// TIA Portal project "Project1500" (V15.1)

(* hardware
DEVICE "S71500/ET200MP station_1"  S7-1500 station
   slot 0: "Rail_0"  Rack  6ES7 590-1***0-0AA0
   slot 1: "PLC_1"  CPU 1515-2 PN  6ES7 515-2AM01-0AB0  V2.6
      slot 3: "CPU display_1"  6ES7591-1BA00-0AA0
*)

// ===== PLC "PLC_1"  CPU 1515-2 PN =====

VAR_GLOBAL   // PLC tag table "Default tag table"
   "Clock_Byte" AT %MB90 : Byte;
   "Clock_10Hz" AT %M90.0 : Bool;
   "Clock_5Hz" AT %M90.1 : Bool;
   "Clock_2.5Hz" AT %M90.2 : Bool;
   "Clock_2Hz" AT %M90.3 : Bool;
   "Clock_1.25Hz" AT %M90.4 : Bool;
   "Clock_1Hz" AT %M90.5 : Bool;
   "Clock_0.625Hz" AT %M90.6 : Bool;
   "Clock_0.5Hz" AT %M90.7 : Bool;
END_VAR

VAR_GLOBAL   // PLC tag table "1AInputs"
   "PLC_AI_CH0" AT %IW64 : Int;   // Резерв
   "PLC_AI_CH1" AT %IW66 : Int;   // Резерв
   "A2_AI_CH0" AT %IW96 : Int;   // Разрежение на газоходе перед циклоном (Элемер-100-ДВ-1231М)
   "A2_AI_CH1" AT %IW98 : Int;   // Разрежение на газоходе перед рукавным фильтром (Элемер-100-ДВ-1231М)
   "A2_AI_CH2" AT %IW100 : Int;   // Разрежение на газоходе после рукавного фильтра (Элемер-100-ДВ-1231М)
   "A2_AI_CH3" AT %IW102 : Int;   // Давление на грубопроводе сжатого воздуха на входе в шатер рукавного фильтра (Элемер-100-ДИ-1150)
   "A2_AI_CH4" AT %IW104 : Int;   // Концентрация CO (Газоанализатор 503б)
   "A2_AI_CH5" AT %IW106 : Int;   // Концентрация SO2 (Газоанализатор 503б)
   "A2_AI_CH6" AT %IW108 : Int;   // Концентрация NOx (Газоанализатор 503б)
   "A2_AI_CH7" AT %IW110 : Int;   // Концентрация CO2 (Газоанализатор 503б)
   "A3_AI_CH0" AT %IW112 : Int;   // Концентрация O2 (Газоанализатор 503б)
   "A3_AI_CH1" AT %IW114 : Int;   // Расход пылегазовой смеси (Анализатор 303в)
   "A3_AI_CH2" AT %IW116 : Int;   // Концентрация пыли (Пылемер 403в)
   "A3_AI_CH3" AT %IW118 : Int;   // Положение: клапан регулирующий для аспирации 1M
   "A3_AI_CH4" AT %IW120 : Int;   // Контроль тока двигателя (Шкаф преобразователя частоты ШПЧ1)
   "A3_AI_CH5" AT %IW122 : Int;   // Контроль скорости двигателя (Шкаф преобразователя частоты ШПЧ1)
   "A3_AI_CH6" AT %IW124 : Int;   // Резерв
   "A3_AI_CH7" AT %IW126 : Int;   // Резерв
   "A4_AI_CH0" AT %IW128 : Int;   // Дымосос 1. Вибрация переднего подшипника вентилятора X-направления
   "A4_AI_CH1" AT %IW130 : Int;   // Дымосос 1. Вибрация переднего подшипника вентилятора Y-направления
   "A4_AI_CH2" AT %IW132 : Int;   // Дымосос 1. Вибрация заднего подшипника вентилятора X-направления
   "A4_AI_CH3" AT %IW134 : Int;   // Дымосос 1. Вибрация заднего подшипника вентилятора Y-направления
   "A4_AI_CH4" AT %IW136 : Int;   // Резерв
   "A4_AI_CH5" AT %IW138 : Int;   // Резерв
   "A4_AI_CH6" AT %IW140 : Int;   // Резерв
   "A4_AI_CH7" AT %IW142 : Int;   // Резерв
   "A5_AI_CH0" AT %IW144 : Int;   // Дымосос 1. Температура переднего подшипника вентилятора (Термопреобр. сопротивления TC-1088-Pt100)
   "A5_AI_CH1" AT %IW146 : Int;   // Дымосос 1. Температура заднего подшипника вентилятора (Термопреобр. сопротивления TC-1088-Pt100)
   "A5_AI_CH2" AT %IW148 : Int;   // Электродвигатель дымососа 1. Температура переднего подшипника (Термопреобр. сопротивления TC-1088-Pt100)
   "A5_AI_CH3" AT %IW150 : Int;   // Электродвигатель дымососа 1. Температура заднего подшипника (Термопреобр. сопротивления TC-1088-Pt100)
   "A5_AI_CH4" AT %IW152 : Int;   // Электродвигатель дымососа 1. Температура обмотки А (Термопреобр. сопротивления TC-1088-Pt100)
   "A5_AI_CH5" AT %IW154 : Int;   // Электродвигатель дымососа 1. Температура обмотки А' (Термопреобр. сопротивления TC-1088-Pt100)
   "A5_AI_CH6" AT %IW156 : Int;   // Электродвигатель дымососа 1. Температура обмотки B (Термопреобр. сопротивления TC-1088-Pt100)
   "A5_AI_CH7" AT %IW158 : Int;   // Электродвигатель дымососа 1. Температура обмотки B' (Термопреобр. сопротивления TC-1088-Pt100)
   "A6_AI_CH0" AT %IW160 : Int;   // Электродвигатель дымососа 1. Температура обмотки C (Термопреобр. сопротивления TC-1088-Pt100)
   "A6_AI_CH1" AT %IW162 : Int;   // Электродвигатель дымососа 1. Температура обмотки C' (Термопреобр. сопротивления TC-1088-Pt100)
   "A6_AI_CH2" AT %IW164 : Int;   // Резерв
   "A6_AI_CH3" AT %IW166 : Int;   // Резерв
   "A6_AI_CH4" AT %IW168 : Int;   // Температура на газоходе перед циклоном (Термопреобр. сопротивления TC-1088-Pt100)
   "A6_AI_CH5" AT %IW170 : Int;   // Температура на газоходе перед рукавным фильтром (Термопреобр. сопротивления TC-1088-Pt100)
   "A6_AI_CH6" AT %IW172 : Int;   // Температура газа на выходе из трубы (Термопреобр. сопротивления TC-1088-Pt100)
   "A6_AI_CH7" AT %IW174 : Int;   // Резерв
END_VAR

VAR_GLOBAL   // PLC tag table "1DInputs"
   "PLC_DI_CH00" AT %I0.0 : Bool;   // Дискретн.вход от реле 10KV1.Высокое напряжение подано (Шкаф преобразователя частоты ШПЧ1)
   "PLC_DI_CH01" AT %I0.1 : Bool;   // Дискретн.вход от реле 10KV2.Режим МУ (Шкаф преобразователя частоты ШПЧ1)
   "PLC_DI_CH02" AT %I0.2 : Bool;   // Дискретн.вход от реле 10KV5.Режим ДУ (Шкаф преобразователя частоты ШПЧ1)
   "PLC_DI_CH03" AT %I0.3 : Bool;   // Дискретн.вход от реле 10KV6.Разрешить импульсы (Шкаф преобразователя частоты ШПЧ1)
   "PLC_DI_CH04" AT %I0.4 : Bool;   // Дискретн.вход от реле 10KV7.Нет аварии (Шкаф преобразователя частоты ШПЧ1)
   "PLC_DI_CH05" AT %I0.5 : Bool;   // Дискретн.вход от реле 10KV11.Сигнал ГОТОВНОСТЬ (Шкаф преобразователя частоты ШПЧ1)
   "PLC_DI_CH06" AT %I0.6 : Bool;   // Дискретн.вход от реле 10KV13.Дистанционное управление (Шкаф преобразователя частоты ШПЧ1)
   "PLC_DI_CH07" AT %I0.7 : Bool;   // Дискретн.вход от реле 10KV14.Местное управление (Шкаф преобразователя частоты ШПЧ1)
   "PLC_DI_CH08" AT %I1.0 : Bool;   // Резерв
   "PLC_DI_CH09" AT %I1.1 : Bool;   // Резерв
   "PLC_DI_CH10" AT %I1.2 : Bool;   // Резерв
   "PLC_DI_CH11" AT %I1.3 : Bool;   // Резерв
   "PLC_DI_CH12" AT %I1.4 : Bool;   // Резерв
   "PLC_DI_CH13" AT %I1.5 : Bool;   // Резерв
   "A7_DI_CH00" AT %I28.0 : Bool;   // Дискретн. вход от реле 2KV1. Направляющий аппарат 2М. Напряжение подано
   "A7_DI_CH01" AT %I28.1 : Bool;   // Дискретн. вход от реле 2KV4. Направляющий аппарат 2М. Выбран режим ДУ
   "A7_DI_CH02" AT %I28.2 : Bool;   // Дискретн. вход от реле 2KM. Направляющий аппарат 2М. Сигнал РАБОТА
   "A7_DI_CH03" AT %I28.3 : Bool;   // Дискретн. вход от реле 2KV2. Направляющий аппарат 2М.Полностью ОТКРЫТ
   "A7_DI_CH04" AT %I28.4 : Bool;   // Дискретн. вход от реле 2KV3. Направляющий аппарат 2М.Полностью ЗАКРЫТ
   "A7_DI_CH05" AT %I28.5 : Bool;   // Дискретн. вход от реле 3KV1. Затвор шлюзовый 3М. Напряжение подано
   "A7_DI_CH06" AT %I28.6 : Bool;   // Дискретн. вход от реле 3KV2. Затвор шлюзовый 3М. Выбран режим ДУ
   "A7_DI_CH07" AT %I28.7 : Bool;   // Дискретн. вход от реле 3KM1. Затвор шлюзовый 3М. Сигнал РАБОТА
   "A7_DI_CH08" AT %I29.0 : Bool;   // Дискретн. вход от реле 1KV8. Клапан регулирующий для аспирации 1М. Напряжение подано
   "A7_DI_CH09" AT %I29.1 : Bool;   // Дискретн. вход от реле 1KV6. Клапан регулирующий для аспирации 1М. Выбран режим ДУ
   "A7_DI_CH10" AT %I29.2 : Bool;   // Дискретн. вход от реле 1KМ1 и 1KV8. Клапан регулирующий 1М. Сигнал ГОТОВНОСТЬ
   "A7_DI_CH11" AT %I29.3 : Bool;   // Дискретн. вход от реле 1KV3. Клапан регулирующий для аспирации 1М. Полностью ОТКРЫТ
   "A7_DI_CH12" AT %I29.4 : Bool;   // Дискретн. вход от реле 1KV4. Клапан регулирующий для аспирации 1М. Полностью ЗАКРЫТ
   "A7_DI_CH13" AT %I29.5 : Bool;   // Дискретн. вход от реле 4KV1. Затвор шлюзовый 4М. Напряжение подано
   "A7_DI_CH14" AT %I29.6 : Bool;   // Дискретн. вход от реле 4KV2. Затвор шлюзовый 4М. Выбран режим ДУ
   "A7_DI_CH15" AT %I29.7 : Bool;   // Дискретн. вход от реле 4KM1. Затвор шлюзовый 4М. Сигнал РАБОТА
   "A8_DI_CH00" AT %I32.0 : Bool;   // Дискретн. вход от реле 5KV1. Затвор шлюзовый 5М. Напряжение подано
   "A8_DI_CH01" AT %I32.1 : Bool;   // Дискретн. вход от реле 5KV2. Затвор шлюзовый 5М. Режим ДУ
   "A8_DI_CH02" AT %I32.2 : Bool;   // Дискретн. вход от реле 5KM1. Затвор шлюзовый 5М. Сигнал РАБОТА
   "A8_DI_CH03" AT %I32.3 : Bool;   // Дискретн. вход от реле 6KV1. Затвор шлюзовый 6М. Напряжение подано
   "A8_DI_CH04" AT %I32.4 : Bool;   // Дискретн. вход от реле 6KV2. Затвор шлюзовый 6М. Режим ДУ
   "A8_DI_CH05" AT %I32.5 : Bool;   // Дискретн. вход от реле 6KM1. Затвор шлюзовый 6М. Сигнал РАБОТА
   "A8_DI_CH06" AT %I32.6 : Bool;   // Резерв
   "A8_DI_CH07" AT %I32.7 : Bool;   // Резерв
   "A8_DI_CH08" AT %I33.0 : Bool;   // Дискретн. вход от реле 7KV1. Затвор шлюзовый 7М. Напряжение подано
   "A8_DI_CH09" AT %I33.1 : Bool;   // Дискретн. вход от реле 7KV2. Затвор шлюзовый 7М. Режим ДУ
   "A8_DI_CH10" AT %I33.2 : Bool;   // Дискретн. вход от реле 7KM1. Затвор шлюзовый 7М. Сигнал РАБОТА
   "A8_DI_CH11" AT %I33.3 : Bool;   // Дискретн. вход от реле 8KV1. Затвор шлюзовый 8М. Напряжение подано
   "A8_DI_CH12" AT %I33.4 : Bool;   // Дискретн. вход от реле 8KV2. Затвор шлюзовый 8М. Режим ДУ
   "A8_DI_CH13" AT %I33.5 : Bool;   // Дискретн. вход от реле 8KM1. Затвор шлюзовый 8М. Сигнал РАБОТА
   "A8_DI_CH14" AT %I33.6 : Bool;   // Резерв
   "A8_DI_CH15" AT %I33.7 : Bool;   // Резерв
   "A9_DI_CH00" AT %I36.0 : Bool;   // Ввод-1 230В, 50Гц вводной выключатель ШЭ - включен (Шкаф электроснабжения (ШЭ)
   "A9_DI_CH01" AT %I36.1 : Bool;   // Фидер 230В, 50Гц 1ШК ФРИР Включен - Питание клапанов (Шкаф электроснабжения (ШЭ)
   "A9_DI_CH02" AT %I36.2 : Bool;   // 230В, 50Гц Выключатель ИБП Выключен (Шкаф электроснабжения (ШЭ)
   "A9_DI_CH03" AT %I36.3 : Bool;   // Фидер 230В, 50Гц 1ШК ФРИР от ИБП Включен - Питание ПЛК, датчиков (Шкаф электроснабжения (ШЭ)
   "A9_DI_CH04" AT %I36.4 : Bool;   // Фидер 230В, 50Гц 1ШК ГО от ИБП Включен
   "A9_DI_CH05" AT %I36.5 : Bool;   // Фидер 230В, 50Гц ШГМ от ИБП Включен
   "A9_DI_CH06" AT %I36.6 : Bool;   // Фидер 230В, 50Гц ШРС от ИБП Включен
   "A9_DI_CH07" AT %I36.7 : Bool;   // Вводный выключатель обогрева шкафа ШЭ включен
   "A9_DI_CH08" AT %I37.0 : Bool;   // В норме - Контроль уровня заряда батареи (Шкаф электроснабж.ШЭ)
   "A9_DI_CH09" AT %I37.1 : Bool;   // Ниже допустимого - Контроль уровня заряда батареи (Шкаф электроснабж.ШЭ)
   "A9_DI_CH10" AT %I37.2 : Bool;   // Дверь ШЭ закрыта при подкл. Агрегате к питанию 230В,50Гц -контакт К2 замкнут. (Шкаф электроснабж.ШЭ)
   "A9_DI_CH11" AT %I37.3 : Bool;   // Вводный выключатель кондиционера ШЭ включен (Шкаф электроснабж.ШЭ)
   "A9_DI_CH12" AT %I37.4 : Bool;   // Дверь 1ШК ГО закрыта при подкл.агрегате к питанию 230В,50Гц (Контакт К2 замкнут)
   "A9_DI_CH13" AT %I37.5 : Bool;   // Температура в 1ШК ГО при подкл.агрегата к питанию 230В,50Гц в норме-контакт К1 замкнут. (Шкаф электроснабж.ШЭ)
   "A9_DI_CH14" AT %I37.6 : Bool;   // Температура в ШЭ при подкл. агрегате к питанию ~230В,50Гц в норме (контакт К1 замкнут)
   "A9_DI_CH15" AT %I37.7 : Bool;   // Резерв
END_VAR

VAR_GLOBAL   // PLC tag table "1Merckers"
   "xFirstStep" AT %M99.7 : Bool;   // Признак первого цикла программы
   "xSimulation" AT %M99.0 : Bool;   // Симуляция включена
   "xTrue" AT %M99.1 : Bool;   // Логическая единица
   "x1M_Output_DN" AT %M1.0 : Bool;   // Команда DN от ПИД-регулятора для 1М
   "xSelectErrRange" AT %M99.2 : Bool;   // Выбор диапазона для ошибки канала аналогоаого входа
   "iValueErrRangeMin" AT %MW100 : Int;   // Минимум кода АЦП для ошибки канала аналогоаого входа
   "iValueErrRangeMax" AT %MW102 : Int;   // Максимум кода АЦП для ошибки канала аналогоаого входа
   "iDeltaErrRangeUp" AT %MW104 : Int;   // Смещение вверх кода АЦП для ошибки канала аналогоаого входа
   "x1000ms" AT %M99.3 : Bool;   // Признак новой секунды
   "iDeltaErrRangeDown" AT %MW106 : Int;   // Смещение вниз кода АЦП для ошибки канала аналогоаого входа
   "xReset1M" AT %M77.1 : Bool;   // Перезапуск ПИДа 1М
   "x1M_Output_UP" AT %M1.1 : Bool;   // Команда UP от ПИД-регулятора для 1М
   "x2M_AutoModeCommand" AT %M2.2 : Bool;   // Команда авт.режима Управлять для 2М
   "x8M_AutoModeCommand" AT %M8.2 : Bool;   // Команда авт.режима Включить для 8М. Не исп.
   "x7M_AutoModeCommand" AT %M7.2 : Bool;   // Команда авт.режима Включить для 7М. Не исп.
   "x3M_AutoModeCommand" AT %M3.2 : Bool;   // Команда авт.режима Включить для 3М. Не исп.
   "x4M_AutoModeCommand" AT %M4.2 : Bool;   // Команда авт.режима Включить для 4М. Не исп.
   "x5M_AutoModeCommand" AT %M5.2 : Bool;   // Команда авт.режима Включить для 5М. Не исп.
   "x6M_AutoModeCommand" AT %M6.2 : Bool;   // Команда авт.режима Включить для 6М. Не исп.
   "iDymPID_Command" AT %MW10 : Int;   // Задание скорости приводу дымососа от ПИДа
   "xResetDym" AT %M77.2 : Bool;   // Перезапуск ПИДа дымососа
   "x2M_AutoModeOpen" AT %M2.3 : Bool;   // Команда авт.режима Открыть для 2М
   "x2M_AutoModeClose" AT %M2.4 : Bool;   // Команда авт.режима Закрыть для 2М
   "xInterlocks" AT %M99.4 : Bool;   // Для активации передачи на ФРИР
   "xNewHour" AT %M99.5 : Bool;   // Признак нового часа
   "iHourOld" AT %MB86 : USInt;   // Старый час системного времени
   "xNULL" AT %M0.0 : Bool;   // Это если функция выдает статус, но он не исп.
   "timBefNH" AT %MD82 : Time;   // Осталось времени до нового часа
   "rMotorSpeed" AT %MD12 : Real;   // Скорость двигателя дымососа в %
   "xFirstSecond" AT %M99.6 : Bool;   // Признак первого прохода циклической программы 1000ms
   "iMinuteOld" AT %MB87 : USInt;   // Старая минута системного времени
   "usiBefMin" AT %MB80 : USInt;   // Осталось минут до нового часа
   "usiBefSec" AT %MB81 : USInt;   // Осталось секунд до нового часа
   "rMotorCurrent" AT %MD16 : Real;   // Ток двигателя дымососа в %
   "xAlarmSirenOn" AT %M98.6 : Bool;   // Включить звуковую сигнализацию
   "xAlarmLampOn" AT %M98.7 : Bool;   // Включить световую сигнализацию
   "iAlarmCount" AT %MW96 : Int;   // Счетчик аварий
   "iAlarmCountOld" AT %MW94 : Int;   // Счетчик аварий на предыдущем проходе
   "x1M_Ready" AT %M20.1 : Bool;   // Готовность
   "xDymReady" AT %M20.0 : Bool;   // Готовность дымососа
   "x2M_Ready" AT %M20.2 : Bool;   // Готовность
   "x3M_Ready" AT %M20.3 : Bool;   // Готовность
   "x4M_Ready" AT %M20.4 : Bool;   // Готовность
   "x5M_Ready" AT %M20.5 : Bool;   // Готовность
   "x6M_Ready" AT %M20.6 : Bool;   // Готовность
   "x7M_Ready" AT %M20.7 : Bool;   // Готовность
   "x8M_Ready" AT %M21.0 : Bool;   // Готовность
END_VAR

VAR_GLOBAL   // PLC tag table "1Outputs"
   "PLC_AO_CH0" AT %QW64 : Int;   // Код ЦАП аналогов. выхода RV1 Задание скорости (Шкаф ШПЧ1)
   "PLC_AO_CH1" AT %QW66 : Int;   // Резерв
   "PLC_DO_CH00" AT %Q0.0 : Bool;   // Резерв
   "PLC_DO_CH01" AT %Q0.1 : Bool;   // Резерв
   "PLC_DO_CH02" AT %Q0.2 : Bool;   // Резерв
   "PLC_DO_CH03" AT %Q0.3 : Bool;   // Резерв
   "PLC_DO_CH04" AT %Q0.4 : Bool;   // Резерв
   "PLC_DO_CH05" AT %Q0.5 : Bool;   // Резерв
   "PLC_DO_CH06" AT %Q0.6 : Bool;   // Резерв
   "PLC_DO_CH07" AT %Q0.7 : Bool;   // Резерв
   "PLC_DO_CH08" AT %Q1.0 : Bool;   // Резерв
   "PLC_DO_CH09" AT %Q1.1 : Bool;   // Резерв
   "A7_DO_CH00" AT %Q28.0 : Bool;   // Дискретн. выход катушки реле 2KV5. Команда ОТКРЫТЬ (Направляющий аппарат 2М)
   "A7_DO_CH01" AT %Q28.1 : Bool;   // Дискретн. выход катушки реле 2KV6. Команда ЗАКРЫТЬ (Направляющий аппарат 2М)
   "A7_DO_CH02" AT %Q28.2 : Bool;   // Дискретн. выход катушки реле 1KV2. Команда ОТКРЫТЬ (Регулирующий клапан 1М)
   "A7_DO_CH03" AT %Q28.3 : Bool;   // Дискретн. выход катушки реле 1KV1. Команда ЗАКРЫТЬ (Регулирующий клапан 1М)
   "A7_DO_CH04" AT %Q28.4 : Bool;   // Дискретн. выход катушки реле 3KV3. Команда ПУСК (Затвор шлюзовый 3М)
   "A7_DO_CH05" AT %Q28.5 : Bool;   // Дискретн. выход катушки реле 4KV3. Команда ПУСК (Затвор шлюзовый 4М)
   "A7_DO_CH06" AT %Q28.6 : Bool;   // Дискретн. выход катушки реле 5KV3. Команда ПУСК (Затвор шлюзовый 5М)
   "A7_DO_CH07" AT %Q28.7 : Bool;   // Дискретн. выход катушки реле 6KV3. Команда ПУСК (Затвор шлюзовый 6М)
   "A7_DO_CH08" AT %Q29.0 : Bool;   // Дискретн. выход катушки реле 7KV3. Команда ПУСК (Затвор шлюзовый 7М)
   "A7_DO_CH09" AT %Q29.1 : Bool;   // Дискретн. выход катушки реле 8KV3. Команда ПУСК (Затвор шлюзовый 8М)
   "A7_DO_CH10" AT %Q29.2 : Bool;   // Дискретн. выход катушки реле 10KV9. Команда ПУСК (ШПЧ1)
   "A7_DO_CH11" AT %Q29.3 : Bool;   // Дискретн. выход катушки реле 10KV10.Команда СТОП (ШПЧ1)
   "A7_DO_CH12" AT %Q29.4 : Bool;   // Резерв
   "A7_DO_CH13" AT %Q29.5 : Bool;   // Резерв
   "A7_DO_CH14" AT %Q29.6 : Bool;   // Дискретн. выход Аварийная сигнализация, звонок
   "A7_DO_CH15" AT %Q29.7 : Bool;   // Дискретн. выход Аварийная сигнализация, лампа
   "A8_DO_CH00" AT %Q32.0 : Bool;   // Резерв
   "A8_DO_CH01" AT %Q32.1 : Bool;   // Резерв
   "A8_DO_CH02" AT %Q32.2 : Bool;   // Резерв
   "A8_DO_CH03" AT %Q32.3 : Bool;   // Резерв
   "A8_DO_CH04" AT %Q32.4 : Bool;   // Резерв
   "A8_DO_CH05" AT %Q32.5 : Bool;   // Резерв
   "A8_DO_CH06" AT %Q32.6 : Bool;   // Резерв
   "A8_DO_CH07" AT %Q32.7 : Bool;   // Резерв
   "A8_DO_CH08" AT %Q33.0 : Bool;   // Резерв
   "A8_DO_CH09" AT %Q33.1 : Bool;   // Резерв
   "A8_DO_CH10" AT %Q33.2 : Bool;   // Резерв
   "A8_DO_CH11" AT %Q33.3 : Bool;   // Резерв
   "A8_DO_CH12" AT %Q33.4 : Bool;   // Резерв
   "A8_DO_CH13" AT %Q33.5 : Bool;   // Резерв
   "A8_DO_CH14" AT %Q33.6 : Bool;   // Резерв
   "A8_DO_CH15" AT %Q33.7 : Bool;   // Резерв
   "A9_DO_CH00" AT %Q36.0 : Bool;   // Резерв
   "A9_DO_CH01" AT %Q36.1 : Bool;   // Резерв
   "A9_DO_CH02" AT %Q36.2 : Bool;   // Резерв
   "A9_DO_CH03" AT %Q36.3 : Bool;   // Резерв
   "A9_DO_CH04" AT %Q36.4 : Bool;   // Резерв
   "A9_DO_CH05" AT %Q36.5 : Bool;   // Резерв
   "A9_DO_CH06" AT %Q36.6 : Bool;   // Резерв
   "A9_DO_CH07" AT %Q36.7 : Bool;   // Резерв
   "A9_DO_CH08" AT %Q37.0 : Bool;   // Резерв
   "A9_DO_CH09" AT %Q37.1 : Bool;   // Резерв
   "A9_DO_CH10" AT %Q37.2 : Bool;   // Резерв
   "A9_DO_CH11" AT %Q37.3 : Bool;   // Резерв
   "A9_DO_CH12" AT %Q37.4 : Bool;   // Резерв
   "A9_DO_CH13" AT %Q37.5 : Bool;   // Резерв
   "A9_DO_CH14" AT %Q37.6 : Bool;   // Резерв
   "A9_DO_CH15" AT %Q37.7 : Bool;   // Резерв
END_VAR

TYPE "uScale"
   STRUCT
      Xmax : Int := 27648;   // Верхняя граница кода АЦП
      Xmin : Int := 0;   // Нижняя граница кода АЦП
      Qmax : Real := 100.0;   // Конец шкалы. Верхняя граница физического диапазона
      Qmin : Real := 0.0;   // Начало шкалы. Нижняя граница физического диапазона
      LimitOn : Bool := false;   // Включение лимитирования
      FilterON : Bool := true;   // Включение фильтра
      FilterTau : Real := 1.0;   // Время фильтрации, сек
   END_STRUCT;
END_TYPE

TYPE "uWrnngAlarm"
   STRUCT
      H : Real;   // Уставка верхнего предела сигнализации
      L : Real;   // Уставка нижнего предела сигнализации
      Delay : Time := t#3s;   // Задержка на срабатывание
      HighOn : Bool;   // Достигнут верхний предел сигнализации
      LowOn : Bool;   // Достигнут нижний предел сигнализации
      H_switch : Bool;   // Активация сигнализации верхнего лимита
      L_switch : Bool;   // Активация сигнализации нижнего лимита
   END_STRUCT;
END_TYPE

TYPE "uHMI-PID"
   STRUCT
      rSetpoint : Real;   // Уставка ПИД-регулятора в обычном режиме [физ.ед]
      rProportionalGain : Real;   // Коэффициент прпорционального усиления
      rIntegralActionTime : Real;   // Время интегрирования [сек]
      rDerivativeActionTime : Real;   // Время дифференцирования [сек]
      rDeadbandWidth : Real;   // Зона нечувствительности [физ.ед]
      r6 : Real;
      r7 : Real;
      r8 : Real;
      rPID_GoTo : Real := 10.0;   // Уставка ПИД-регулятора для режима перемещения в заданное положение [%]
      i10 : Int;
      spare0 : Bool;
      spare1 : Bool;
      spare2 : Bool;
      spare3 : Bool;
      xSwitchPID_Mode : Bool;   // 0-обычный, 1-заданное положение
      spare5 : Bool;
      spare6 : Bool;
      spare7 : Bool;
      spare8 : Bool;
   END_STRUCT;
END_TYPE

TYPE "uHMI-Machine"
   STRUCT
      rPosition : Real;   // Положение/позиция механизма [физ.ед]
      rPosGoTo : Real := 10.0;   // Уставка перемещения в заданное положение [%]
      Spare_R : Real;
      wMode : UInt;   // Режим управления механизмом
      wPositionCode : UInt;   // Код положения механизма
      wStatusCode : UInt;   // Статус/состояние механизма
      wCommandCode : UInt;   // Код управления механизмом
      wWarnings : Word;   // Предупреждения
      wAlarms : Word;   // Аварии
      Spare_26 : Word;
      Spare_28 : Word;
      xReady : Bool;   // Готовность механизма
      xButManOpen : Bool;   // Кнопка на ручное открытие
      xButManClose : Bool;   // Кнопка на ручное закрытие
      xButtonGoTo : Bool;   // Кнопка Перемещение В Заданное Положение
      xSwitchAutoMode : Bool;   // Переключатель автоматический / ручной на ЧМИ
      xButtonAck : Bool;   // Сброс аварии механизма
      Spare_06 : Bool;
      Spare_07 : Bool;
      Spare_08 : Bool;
      Spare_09 : Bool;
      Spare_10 : Bool;
      Spare_11 : Bool;
      Spare_12 : Bool;
      Spare_13 : Bool;
      Spare_14 : Bool;
      Spare_15 : Bool;
   END_STRUCT;
END_TYPE

TYPE "uHMI-Dym"
   STRUCT
      rSpeed : Real;   // Скорость двигателя
      rSpeedGoTo : Real := 10.0;   // Уставка для ручного задания скорости
      timBackCount : Time;   // Таймер обратного отсчета, если пуски исчерпаны
      wMode : UInt;   // Режим управления механизмом
      wPositionCode : UInt;   // Код положения механизма
      wStatusCode : UInt;   // Статус/состояние механизма
      wCommandCode : UInt;   // Код управления механизмом
      wWarnings : Word;   // Предупреждения
      wAlarms : Word;   // Аварии
      iMaxStart : Int;   // Максимальное число пусков в час
      iNumStart : Int;   // Текущее число пусков в час
      xReady : Bool;   // Готовность механизма
      xButStart : Bool;   // Кнопка СТАРТ
      xButStop : Bool;   // Кнопка СТОП
      xButtonGoTo : Bool;   // Кнопка Установить Скорость ручного режима
      xSwitchAutoMode : Bool;   // Переключатель автоматический / ручной на ЧМИ
      xButtonAck : Bool;   // Сброс аварии механизма
      Spare_06 : Bool;
      Spare_07 : Bool;
      xReadyMaxStart : Bool;   // Готовность по числу пусков в час
      Spare_09 : Bool;
      Spare_10 : Bool;
      Spare_11 : Bool;
      Spare_12 : Bool;
      Spare_13 : Bool;
      Spare_14 : Bool;
      Spare_15 : Bool;
   END_STRUCT;
END_TYPE

// folder: Simulation

TYPE "uAI"
   STRUCT
      Value_nepr : Real;   // Значение / Неприведенный (если расход газа)
      Value : Real;   // Значение / Значение в физ. единицах
      Value_filtr : Real;   // Значение в физ. единицах после фильтра
      mA : Real;   // Ток / Ток канала в mA
      Min : Real;   // Минимум шкалы / Начало шкалы
      NAG : Real;   // Нижняя аварийная граница
      NPG : Real;   // Нижняя предупредительная граница
      VPG : Real;   // Верхняя предупредительная граница
      VAG : Real;   // Верхняя аварийная граница
      Max : Real;   // Максимум шкалы / Конец шкалы
      Kkorr : Real := 1.0;   // Коэффициент коррекции
      Pnorm : Real;   // Нормальное давление канала
      Tnorm : Real;   // Нормальная температура канала
      Kfiltr : Int;   // Коэффициент фильтра
      Alarm : Word;   // 0-норма,1-НПГ,2-ВПГ,4-НАГ,8-ВАГ,16-внеПред,32-обрыв,64-перегр.
   END_STRUCT;
END_TYPE

TYPE "uSim"
   STRUCT
      config : Struct
         s256 : Bool;
         s512 : Bool;
         s1024 : Bool;
         s2048 : Bool;
         s4096 : Bool;
         s8192 : Bool;
         s16384 : Bool;
         s32768 : Bool;
         down : Bool;   // Симуляция вверх
         up : Bool;   // Симуляция вниз
         auto : Bool;   // Симуляция включена
         s8 : Bool;
         s16 : Bool;
         s32 : Bool;
         s64 : Bool;
         s128 : Bool;
      END_STRUCT;
      factor : Real := 241.0;   // К-т усиления
      offset : Real := 194.0;   // Смещение
      iCounter : Int;   // Счетчик для массива симуляции
      Value : Int;   // Значение мз массива симуляции
      spare1 : Int;
      spare2 : Int;
      spare3 : Int;
   END_STRUCT;
END_TYPE

// folder: (top level)

DATA_BLOCK "1DB_AIConfig"   // DB6
TITLE = Конфигурация аналоговых входов
{ S7_Optimized_Access := 'FALSE' }
VERSION : 0.1
// Блок данных содержит параметры шкалы, фильтрации, признак лимитирования
   VAR
      RarefactFlueInCyclone : "uScale";   // Разрежение на газоходе перед циклоном PIT201a
      RarefactFlueInFilter : "uScale";   // Разрежение на газоходе перед рукавным фильтром PIT202a
      RarefactFlueOutFilter : "uScale";   // Разрежение на газоходе после рукавного фильтра PIT203a
      PressureComprAir : "uScale";   // Давл. на трубопроводе сж.воздуха на вх. в шатер рукавного фильтра PIT204a
      GasAnalyzerCO : "uScale";   // Концентрация CO QT503b_CO
      GasAnalyzerSO2 : "uScale";   // Концентрация SO2 QT503b_SO2
      GasAnalyzerNOx : "uScale";   // Концентрация NOx QT503b_NOx
      GasAnalyzerCO2 : "uScale";   // Концентрация CO2 QT503b_CO2.
      GasAnalyzerO2 : "uScale";   // Концентрация O2 QT503b_O2
      FlowDustGasMix : "uScale";   // Расход пылегазовой смеси QT303b
      GasAnalyzerDust : "uScale";   // Концентрация пыли QT403b
      PosValve1M : "uScale";   // Положение: клапан регулирующий 1M для аспирации PV1M.
      CurrentMotorShPCh1 : "uScale";   // Контроль тока двигателя (Шкаф ШПЧ1) IT1
      RpmMotorShPCh1 : "uScale";   // Контроль скорости (Шкаф ШПЧ1) RT1
      D1FanVibrFrontX : "uScale";   // Дымосос 1. Вибрация переднего подшипника вентилятора X-направления VE801a
      D1FanVibrFrontY : "uScale";   // Дымосос 1. Вибрация переднего подшипника вентилятора Y-направления VE802a
      D1FanVibrBackX : "uScale";   // Дымосос 1. Вибрация заднего подшипника вентилятора X-направления VE803a
      D1FanVibrBackY : "uScale";   // Дымосос 1. Вибрация заднего подшипника вентилятора Y-направления VE804a
      D1FanTempFront : "uScale";   // Дымосос 1. Температура переднего подшипника вентилятора TE104a
      D1FanTempBack : "uScale";   // Дымосос 1. Температура заднего подшипника вентилятора TE105a
      D1MotorTempFront : "uScale";   // Электродвигатель дымососа 1. Температура переднего подшипника TE106a
      D1MotorTempBack : "uScale";   // Электродвигатель дымососа 1. Температура заднего подшипника TE107a
      D1MotorTempWindA1 : "uScale";   // Электродвигатель дымососа 1. Температура обмотки А TE108a
      D1MotorTempWindA2 : "uScale";   // Электродвигатель дымососа 1. Температура обмотки А' TE109a
      D1MotorTempWindB1 : "uScale";   // Электродвигатель дымососа 1. Температура обмотки B TE110a
      D1MotorTempWindB2 : "uScale";   // Электродвигатель дымососа 1. Температура обмотки B TE111a
      D1MotorTempWindC1 : "uScale";   // Электродвигатель дымососа 1. Температура обмотки C TE112a
      D1MotorTempWindC2 : "uScale";   // Электродвигатель дымососа 1. Температура обмотки C' TE113a
      TGasDuctInCyclone : "uScale";   // Температура на газоходе перед циклоном TE101a
      TGasDuctInFilter : "uScale";   // Температура на газоходе перед рукавным фильтром TE102a
      TGasOutPipe : "uScale";   // Температура газа на выходе из трубы TE103a
      uSpare558 : "uScale";   // 1
      uSpare559 : "uScale";   // 2
      uSpare560 : "uScale";   // 3
      uSpare561 : "uScale";   // 4
      uSpare562 : "uScale";   // 5
      uSpare563 : "uScale";   // 6
      uSpare564 : "uScale";   // 7
      uSpare565 : "uScale";   // 8
      uSpare566 : "uScale";   // 9
      uSpare567 : "uScale";   // 10
      uSpare568 : "uScale";   // 11
      uSpare569 : "uScale";   // 12
      uSpare570 : "uScale";   // 13
      uSpare571 : "uScale";   // 14
      uSpare572 : "uScale";   // 15
      uSpare573 : "uScale";   // 16
      uSpare574 : "uScale";   // 17
      "uTest4-20" : "uScale";   // Тестируем алгоритмы Аналогового входа 4-20mA
      uTestRTD : "uScale";   // Тестируем алгоритмы Аналогового входа RTD (термометр)
   END_VAR
BEGIN
   RarefactFlueInCyclone.Qmax := 10.0;
   FlowDustGasMix.Qmax := 500.0;
   RarefactFlueInCyclone.FilterTau := 0.5;
   RarefactFlueInFilter.Qmax := 10.0;
   RarefactFlueOutFilter.Qmax := 10.0;
   PressureComprAir.Qmax := 10.0;
   GasAnalyzerCO.Qmax := 300.0;
   GasAnalyzerSO2.Qmax := 500.0;
   GasAnalyzerNOx.Qmax := 500.0;
   GasAnalyzerCO2.Qmax := 4.0;
   GasAnalyzerO2.Qmax := 20.0;
   GasAnalyzerDust.Qmax := 500.0;
   CurrentMotorShPCh1.Qmax := 906.0;
   RpmMotorShPCh1.Qmax := 991.0;
   D1FanVibrFrontX.Qmax := 20.0;
   D1FanVibrFrontY.Qmax := 20.0;
   D1FanVibrBackX.Qmax := 20.0;
   D1FanVibrBackY.Qmax := 20.0;
   D1FanTempFront.Qmax := 200.0;
   D1FanTempBack.Qmax := 200.0;
   D1MotorTempFront.Qmax := 200.0;
   D1MotorTempBack.Qmax := 200.0;
   D1MotorTempWindA1.Qmax := 200.0;
   D1MotorTempWindA2.Qmax := 200.0;
   D1MotorTempWindB1.Qmax := 200.0;
   D1MotorTempWindB2.Qmax := 200.0;
   D1MotorTempWindC1.Qmax := 200.0;
   D1MotorTempWindC2.Qmax := 200.0;
   TGasDuctInCyclone.Qmax := 350.0;
   TGasDuctInFilter.Qmax := 250.0;
   TGasOutPipe.Qmax := 250.0;
   PosValve1M.FilterON := false;
   RpmMotorShPCh1.FilterTau := 3.0;
   PressureComprAir.FilterTau := 5.0;
   "uTest4-20".LimitOn := 0;
   uTestRTD.LimitOn := 0;
END_DATA_BLOCK

DATA_BLOCK "Scaled_AI"   // DB7
TITLE = Обработанные входные аналоговые сигналы
{ S7_Optimized_Access := 'FALSE' }
VERSION : 0.1
// Блок данных содержит фильтрованные (если установлен признак) физические значения аналоговых сигналов
   VAR
      RarefactFlueInCyclone : Real := 0.0;   // Разрежение на газоходе перед циклоном PIT201a
      RarefactFlueInFilter : Real := 0.0;   // Разрежение на газоходе перед рукавным фильтром PIT202a
      RarefactFlueOutFilter : Real := 0.0;   // Разрежение на газоходе после рукавного фильтра PIT203a
      PressureComprAir : Real := 0.0;   // Давл. на трубопроводе сж.воздуха на вх. в шатер рукавного фильтра PIT204a
      GasAnalyzerCO : Real := 0.0;   // Концентрация CO QT503b_CO
      GasAnalyzerSO2 : Real := 0.0;   // Концентрация SO2 QT503b_SO2
      GasAnalyzerNOx : Real := 0.0;   // Концентрация NOx QT503b_NOx
      GasAnalyzerCO2 : Real := 0.0;   // Концентрация CO2 QT503b_CO2.
      GasAnalyzerO2 : Real := 0.0;   // Концентрация O2 QT503b_O2
      FlowDustGasMix : Real := 0.0;   // Расход пылегазовой смеси QT303b
      GasAnalyzerDust : Real := 0.0;   // Концентрация пыли QT403b
      PosValve1M : Real := 0.0;   // Положение: клапан регулирующий 1M для аспирации PV1M.
      CurrentMotorShPCh1 : Real := 0.0;   // Контроль тока двигателя (Шкаф ШПЧ1) IT1
      RpmMotorShPCh1 : Real := 0.0;   // Контроль скорости (Шкаф ШПЧ1) RT1
      D1FanVibrFrontX : Real := 0.0;   // Дымосос 1. Вибрация переднего подшипника вентилятора X-направления VE801a
      D1FanVibrFrontY : Real := 0.0;   // Дымосос 1. Вибрация переднего подшипника вентилятора Y-направления VE802a
      D1FanVibrBackX : Real := 0.0;   // Дымосос 1. Вибрация заднего подшипника вентилятора X-направления VE803a
      D1FanVibrBackY : Real := 0.0;   // Дымосос 1. Вибрация заднего подшипника вентилятора Y-направления VE804a
      D1FanTempFront : Real := 0.0;   // Дымосос 1. Температура переднего подшипника вентилятора TE104a
      D1FanTempBack : Real := 0.0;   // Дымосос 1. Температура заднего подшипника вентилятора TE105a
      D1MotorTempFront : Real := 0.0;   // Электродвигатель дымососа 1. Температура переднего подшипника TE106a
      D1MotorTempBack : Real := 0.0;   // Электродвигатель дымососа 1. Температура заднего подшипника TE107a
      D1MotorTempWindA1 : Real := 0.0;   // Электродвигатель дымососа 1. Температура обмотки А TE108a
      D1MotorTempWindA2 : Real := 0.0;   // Электродвигатель дымососа 1. Температура обмотки А' TE109a
      D1MotorTempWindB1 : Real := 0.0;   // Электродвигатель дымососа 1. Температура обмотки B TE110a
      D1MotorTempWindB2 : Real := 0.0;   // Электродвигатель дымососа 1. Температура обмотки B TE111a
      D1MotorTempWindC1 : Real := 0.0;   // Электродвигатель дымососа 1. Температура обмотки C TE112a
      D1MotorTempWindC2 : Real := 0.0;   // Электродвигатель дымососа 1. Температура обмотки C' TE113a
      TGasDuctInCyclone : Real := 0.0;   // Температура на газоходе перед циклоном TE101a
      TGasDuctInFilter : Real := 0.0;   // Температура на газоходе перед рукавным фильтром TE102a
      TGasOutPipe : Real := 0.0;   // Температура газа на выходе из трубы TE103a
      rSpare124 : Real;   // 1
      rSpare125 : Real;   // 2
      rSpare126 : Real;   // 3
      rSpare127 : Real;   // 4
      rSpare128 : Real;   // 5
      rSpare129 : Real;   // 6
      rSpare130 : Real;   // 7
      rSpare131 : Real;   // 8
      rSpare132 : Real;   // 9
      rForRegHMI : Real := 4.0;   // Разность разрежений, заданная оператором
      rSpare164 : Real;   // 11
      rSpare165 : Real;   // 12
      rSpare166 : Real;   // 13
      rSpare167 : Real;   // 14
      rSpare168 : Real;   // 15
      rSpare169 : Real;   // 16
      rSpare170 : Real;   // 17
      "rTest4-20" : Real;   // Тестируем алгоритмы Аналогового входа 4-20mA
      rTestRTD : Real;   // Тестируем алгоритмы Аналогового входа RTD (термометр)
   END_VAR
BEGIN
END_DATA_BLOCK

DATA_BLOCK "Alarm_DB"   // DB10
TITLE = Аварийные границы
{ S7_Optimized_Access := 'FALSE' }
VERSION : 0.1
// Блок данных содержит параметры верхней и нижней аварийной границы аналоговых сигналов
   VAR
      RarefactFlueInCyclone : "uWrnngAlarm";   // Разрежение на газоходе перед циклоном PIT201a
      RarefactFlueInFilter : "uWrnngAlarm";   // Разрежение на газоходе перед рукавным фильтром PIT202a
      RarefactFlueOutFilter : "uWrnngAlarm";   // Разрежение на газоходе после рукавного фильтра PIT203a
      PressureComprAir : "uWrnngAlarm";   // Давл. на трубопроводе сж.воздуха на вх. в шатер рукавного фильтра PIT204a
      GasAnalyzerCO : "uWrnngAlarm";   // Концентрация CO QT503b_CO
      GasAnalyzerSO2 : "uWrnngAlarm";   // Концентрация SO2 QT503b_SO2
      GasAnalyzerNOx : "uWrnngAlarm";   // Концентрация NOx QT503b_NOx
      GasAnalyzerCO2 : "uWrnngAlarm";   // Концентрация CO2 QT503b_CO2.
      GasAnalyzerO2 : "uWrnngAlarm";   // Концентрация O2 QT503b_O2
      FlowDustGasMix : "uWrnngAlarm";   // Расход пылегазовой смеси QT303b
      GasAnalyzerDust : "uWrnngAlarm";   // Концентрация пыли QT403b
      PosValve1M : "uWrnngAlarm";   // Положение: клапан регулирующий 1M для аспирации PV1M.
      CurrentMotorShPCh1 : "uWrnngAlarm";   // Контроль тока двигателя (Шкаф ШПЧ1) IT1
      RpmMotorShPCh1 : "uWrnngAlarm";   // Контроль скорости (Шкаф ШПЧ1) RT1
      D1FanVibrFrontX : "uWrnngAlarm";   // Дымосос 1. Вибрация переднего подшипника вентилятора X-направления VE801a
      D1FanVibrFrontY : "uWrnngAlarm";   // Дымосос 1. Вибрация переднего подшипника вентилятора Y-направления VE802a
      D1FanVibrBackX : "uWrnngAlarm";   // Дымосос 1. Вибрация заднего подшипника вентилятора X-направления VE803a
      D1FanVibrBackY : "uWrnngAlarm";   // Дымосос 1. Вибрация заднего подшипника вентилятора Y-направления VE804a
      D1FanTempFront : "uWrnngAlarm";   // Дымосос 1. Температура переднего подшипника вентилятора TE104a
      D1FanTempBack : "uWrnngAlarm";   // Дымосос 1. Температура заднего подшипника вентилятора TE105a
      D1MotorTempFront : "uWrnngAlarm";   // Электродвигатель дымососа 1. Температура переднего подшипника TE106a
      D1MotorTempBack : "uWrnngAlarm";   // Электродвигатель дымососа 1. Температура заднего подшипника TE107a
      D1MotorTempWindA1 : "uWrnngAlarm";   // Электродвигатель дымососа 1. Температура обмотки А TE108a
      D1MotorTempWindA2 : "uWrnngAlarm";   // Электродвигатель дымососа 1. Температура обмотки А' TE109a
      D1MotorTempWindB1 : "uWrnngAlarm";   // Электродвигатель дымососа 1. Температура обмотки B TE110a
      D1MotorTempWindB2 : "uWrnngAlarm";   // Электродвигатель дымососа 1. Температура обмотки B TE111a
      D1MotorTempWindC1 : "uWrnngAlarm";   // Электродвигатель дымососа 1. Температура обмотки C TE112a
      D1MotorTempWindC2 : "uWrnngAlarm";   // Электродвигатель дымососа 1. Температура обмотки C' TE113a
      TGasDuctInCyclone : "uWrnngAlarm";   // Температура на газоходе перед циклоном TE101a
      TGasDuctInFilter : "uWrnngAlarm";   // Температура на газоходе перед рукавным фильтром TE102a
      TGasOutPipe : "uWrnngAlarm";   // Температура газа на выходе из трубы TE103a
      uSpare434 : "uWrnngAlarm";   // 1
      uSpare435 : "uWrnngAlarm";   // 2
      uSpare436 : "uWrnngAlarm";   // 3
      uSpare437 : "uWrnngAlarm";   // 4
      uSpare438 : "uWrnngAlarm";   // 5
      uSpare439 : "uWrnngAlarm";   // 6
      uSpare440 : "uWrnngAlarm";   // 7
      uSpare441 : "uWrnngAlarm";   // 8
      uSpare442 : "uWrnngAlarm";   // 9
      uSpare443 : "uWrnngAlarm";   // 10
      uSpare444 : "uWrnngAlarm";   // 11
      uSpare445 : "uWrnngAlarm";   // 12
      uSpare446 : "uWrnngAlarm";   // 13
      uSpare447 : "uWrnngAlarm";   // 14
      uSpare448 : "uWrnngAlarm";   // 15
      uSpare449 : "uWrnngAlarm";   // 16
      uSpare450 : "uWrnngAlarm";   // 17
      "uTest4-20" : "uWrnngAlarm";   // Тестируем алгоритмы Аналогового входа 4-20mA
      uTestRTD : "uWrnngAlarm";   // Тестируем алгоритмы Аналогового входа RTD (термометр)
   END_VAR
BEGIN
   RarefactFlueInCyclone.H := 5.0;
   RarefactFlueInCyclone.L := 1.0;
   RarefactFlueInFilter.H := 5.0;
   RarefactFlueInFilter.L := 1.0;
   RarefactFlueOutFilter.H := 7.0;
   RarefactFlueOutFilter.H_switch := 1;
   PressureComprAir.H := 0.9;
   PressureComprAir.L := 0.1;
   GasAnalyzerCO.H := 250.0;
   GasAnalyzerCO.H_switch := 1;
   GasAnalyzerSO2.H := 400.0;
   GasAnalyzerSO2.L := 100.0;
   GasAnalyzerNOx.H := 400.0;
   GasAnalyzerNOx.L := 100.0;
   GasAnalyzerCO2.H := 3.5;
   GasAnalyzerCO2.L := 0.5;
   GasAnalyzerO2.H := 18.0;
   GasAnalyzerO2.L := 2.0;
   FlowDustGasMix.H := 400.0;
   FlowDustGasMix.L := 100.0;
   GasAnalyzerDust.H := 400.0;
   GasAnalyzerDust.L := 100.0;
   PosValve1M.H := 90.0;
   PosValve1M.L := 10.0;
   CurrentMotorShPCh1.H := 800.0;
   CurrentMotorShPCh1.L := 100.0;
   RpmMotorShPCh1.H := 800.0;
   RpmMotorShPCh1.L := 100.0;
   D1FanVibrFrontX.H := 18.0;
   D1FanVibrFrontY.H := 18.0;
   D1FanVibrFrontY.H_switch := 1;
   D1FanVibrBackX.H := 18.0;
   D1FanVibrBackX.H_switch := 1;
   D1FanVibrBackY.H := 18.0;
   D1FanVibrBackY.H_switch := 1;
   D1FanTempFront.H := 70.0;
   D1FanTempFront.H_switch := 1;
   D1FanTempBack.H := 70.0;
   D1FanTempBack.H_switch := 1;
   D1MotorTempFront.H := 70.0;
   D1MotorTempFront.H_switch := 1;
   D1MotorTempWindC2.H := 90.0;
   D1MotorTempWindC2.H_switch := 1;
   D1MotorTempWindC1.H := 90.0;
   D1MotorTempWindC1.H_switch := 1;
   D1MotorTempWindB2.H := 90.0;
   D1MotorTempWindB2.H_switch := 1;
   D1MotorTempWindB1.H := 90.0;
   D1MotorTempWindB1.H_switch := 1;
   D1MotorTempWindA2.H := 90.0;
   D1MotorTempWindA2.H_switch := 1;
   D1MotorTempWindA1.H := 90.0;
   D1MotorTempWindA1.H_switch := 1;
   D1MotorTempBack.H := 70.0;
   D1MotorTempBack.H_switch := 1;
   TGasDuctInCyclone.H := 190.0;
   TGasDuctInCyclone.H_switch := 1;
   TGasDuctInFilter.H := 190.0;
   TGasDuctInFilter.H_switch := 1;
   TGasOutPipe.H := 700.0;
   TGasOutPipe.L := 300.0;
   D1FanVibrFrontX.H_switch := 1;
   "uTest4-20".H_switch := 1;
   uTestRTD.H_switch := 1;
   "uTest4-20".H := 85.0;
   "uTest4-20".L := 15.0;
   uTestRTD.H := 85.0;
   uTestRTD.L := 15.0;
END_DATA_BLOCK

DATA_BLOCK "Warning_DB"   // DB15
TITLE = Предупредительные границы
{ S7_Optimized_Access := 'FALSE' }
VERSION : 0.1
// Блок данных содержит параметры верхней и нижней предупредительной границы аналоговых сигналов
   VAR
      RarefactFlueInCyclone : "uWrnngAlarm";   // Разрежение на газоходе перед циклоном PIT201a
      RarefactFlueInFilter : "uWrnngAlarm";   // Разрежение на газоходе перед рукавным фильтром PIT202a
      RarefactFlueOutFilter : "uWrnngAlarm";   // Разрежение на газоходе после рукавного фильтра PIT203a
      PressureComprAir : "uWrnngAlarm";   // Давл. на трубопроводе сж.воздуха на вх. в шатер рукавного фильтра PIT204a
      GasAnalyzerCO : "uWrnngAlarm";   // Концентрация CO QT503b_CO
      GasAnalyzerSO2 : "uWrnngAlarm";   // Концентрация SO2 QT503b_SO2
      GasAnalyzerNOx : "uWrnngAlarm";   // Концентрация NOx QT503b_NOx
      GasAnalyzerCO2 : "uWrnngAlarm";   // Концентрация CO2 QT503b_CO2.
      GasAnalyzerO2 : "uWrnngAlarm";   // Концентрация O2 QT503b_O2
      FlowDustGasMix : "uWrnngAlarm";   // Расход пылегазовой смеси QT303b
      GasAnalyzerDust : "uWrnngAlarm";   // Концентрация пыли QT403b
      PosValve1M : "uWrnngAlarm";   // Положение: клапан регулирующий 1M для аспирации PV1M.
      CurrentMotorShPCh1 : "uWrnngAlarm";   // Контроль тока двигателя (Шкаф ШПЧ1) IT1
      RpmMotorShPCh1 : "uWrnngAlarm";   // Контроль скорости (Шкаф ШПЧ1) RT1
      D1FanVibrFrontX : "uWrnngAlarm";   // Дымосос 1. Вибрация переднего подшипника вентилятора X-направления VE801a
      D1FanVibrFrontY : "uWrnngAlarm";   // Дымосос 1. Вибрация переднего подшипника вентилятора Y-направления VE802a
      D1FanVibrBackX : "uWrnngAlarm";   // Дымосос 1. Вибрация заднего подшипника вентилятора X-направления VE803a
      D1FanVibrBackY : "uWrnngAlarm";   // Дымосос 1. Вибрация заднего подшипника вентилятора Y-направления VE804a
      D1FanTempFront : "uWrnngAlarm";   // Дымосос 1. Температура переднего подшипника вентилятора TE104a
      D1FanTempBack : "uWrnngAlarm";   // Дымосос 1. Температура заднего подшипника вентилятора TE105a
      D1MotorTempFront : "uWrnngAlarm";   // Электродвигатель дымососа 1. Температура переднего подшипника TE106a
      D1MotorTempBack : "uWrnngAlarm";   // Электродвигатель дымососа 1. Температура заднего подшипника TE107a
      D1MotorTempWindA1 : "uWrnngAlarm";   // Электродвигатель дымососа 1. Температура обмотки А TE108a
      D1MotorTempWindA2 : "uWrnngAlarm";   // Электродвигатель дымососа 1. Температура обмотки А' TE109a
      D1MotorTempWindB1 : "uWrnngAlarm";   // Электродвигатель дымососа 1. Температура обмотки B TE110a
      D1MotorTempWindB2 : "uWrnngAlarm";   // Электродвигатель дымососа 1. Температура обмотки B TE111a
      D1MotorTempWindC1 : "uWrnngAlarm";   // Электродвигатель дымососа 1. Температура обмотки C TE112a
      D1MotorTempWindC2 : "uWrnngAlarm";   // Электродвигатель дымососа 1. Температура обмотки C' TE113a
      TGasDuctInCyclone : "uWrnngAlarm";   // Температура на газоходе перед циклоном TE101a
      TGasDuctInFilter : "uWrnngAlarm";   // Температура на газоходе перед рукавным фильтром TE102a
      TGasOutPipe : "uWrnngAlarm";   // Температура газа на выходе из трубы TE103a
      uSpare434 : "uWrnngAlarm";   // 1
      uSpare435 : "uWrnngAlarm";   // 2
      uSpare436 : "uWrnngAlarm";   // 3
      uSpare437 : "uWrnngAlarm";   // 4
      uSpare438 : "uWrnngAlarm";   // 5
      uSpare439 : "uWrnngAlarm";   // 6
      uSpare440 : "uWrnngAlarm";   // 7
      uSpare441 : "uWrnngAlarm";   // 8
      uSpare442 : "uWrnngAlarm";   // 9
      uSpare443 : "uWrnngAlarm";   // 10
      uSpare444 : "uWrnngAlarm";   // 11
      uSpare445 : "uWrnngAlarm";   // 12
      uSpare446 : "uWrnngAlarm";   // 13
      uSpare447 : "uWrnngAlarm";   // 14
      uSpare448 : "uWrnngAlarm";   // 15
      uSpare449 : "uWrnngAlarm";   // 16
      uSpare450 : "uWrnngAlarm";   // 17
      "uTest4-20" : "uWrnngAlarm";   // Тестируем алгоритмы Аналогового входа 4-20mA
      uTestRTD : "uWrnngAlarm";   // Тестируем алгоритмы Аналогового входа RTD (термометр)
   END_VAR
BEGIN
   RarefactFlueInFilter.H := 4.0;
   RarefactFlueInFilter.L := 2.0;
   RarefactFlueInCyclone.H := 4.0;
   RarefactFlueInCyclone.L := 2.0;
   RarefactFlueOutFilter.H := 6.0;
   RarefactFlueOutFilter.H_switch := 1;
   PressureComprAir.H := 0.8;
   PressureComprAir.L := 0.2;
   GasAnalyzerCO.H := 200.0;
   GasAnalyzerCO.H_switch := 1;
   GasAnalyzerSO2.H := 300.0;
   GasAnalyzerSO2.L := 200.0;
   GasAnalyzerNOx.H := 300.0;
   GasAnalyzerNOx.L := 200.0;
   GasAnalyzerCO2.H := 3.0;
   GasAnalyzerCO2.L := 1.0;
   TGasOutPipe.H := 600.0;
   TGasOutPipe.L := 400.0;
   TGasDuctInFilter.H := 180.0;
   TGasDuctInCyclone.H := 180.0;
   TGasDuctInCyclone.H_switch := 1;
   D1MotorTempWindC2.H := 80.0;
   D1MotorTempWindC2.H_switch := 1;
   D1MotorTempWindC1.H := 80.0;
   D1MotorTempWindC1.H_switch := 1;
   D1MotorTempWindB2.H := 80.0;
   D1MotorTempWindB2.H_switch := 1;
   D1MotorTempWindB1.H := 80.0;
   D1MotorTempWindB1.H_switch := 1;
   D1MotorTempWindA2.H := 80.0;
   D1MotorTempWindA2.H_switch := 1;
   D1MotorTempWindA1.H := 80.0;
   D1MotorTempWindA1.H_switch := 1;
   D1MotorTempBack.H := 60.0;
   D1MotorTempBack.H_switch := 1;
   D1MotorTempFront.H := 60.0;
   D1MotorTempFront.H_switch := 1;
   D1FanTempBack.H := 60.0;
   D1FanTempBack.H_switch := 1;
   D1FanTempFront.H := 60.0;
   D1FanTempFront.H_switch := 1;
   D1FanVibrBackY.H := 15.0;
   D1FanVibrBackY.H_switch := 1;
   D1FanVibrBackX.H := 15.0;
   D1FanVibrBackX.H_switch := 1;
   D1FanVibrFrontY.H := 15.0;
   D1FanVibrFrontY.H_switch := 1;
   D1FanVibrFrontX.H := 15.0;
   D1FanVibrFrontX.H_switch := 1;
   RpmMotorShPCh1.H := 700.0;
   RpmMotorShPCh1.L := 200.0;
   CurrentMotorShPCh1.H := 700.0;
   CurrentMotorShPCh1.L := 200.0;
   PosValve1M.H := 80.0;
   PosValve1M.L := 20.0;
   GasAnalyzerDust.H := 300.0;
   GasAnalyzerDust.L := 200.0;
   FlowDustGasMix.H := 300.0;
   FlowDustGasMix.L := 200.0;
   GasAnalyzerO2.H := 15.0;
   GasAnalyzerO2.L := 5.0;
   TGasDuctInFilter.H_switch := 1;
   uTestRTD.H_switch := 1;
   uTestRTD.H := 70.0;
   uTestRTD.L := 30.0;
   "uTest4-20".H := 70.0;
   "uTest4-20".L := 30.0;
   "uTest4-20".H_switch := 1;
END_DATA_BLOCK

DATA_BLOCK "1DB_Communication"   // DB100
{ S7_Optimized_Access := 'FALSE' }
VERSION : 0.1
   VAR
      xRegDeltaP : Bool;   // Сигнал передается во ФРИР для регенерации рукавного фильтра
      xTotalSTOP : Bool;   // Функциональный останов для ФРИР
      wWord2 : Word;
      wWord3 : Word;
      wWord4 : Word;
      wFrom1to2 : UInt;   // Инкремент каждые 0.8сек для состояния связи
      xSpare7 : Bool;
      xSpare8 : Bool;
      xSpare9 : Bool;
      x3MfromLevel : Bool;   // Управление затвором 3М в автомат.режиме
      x4MfromLevel : Bool;   // Управление затвором 4М в автомат.режиме
      x5MfromLevel : Bool;   // Управление затвором 5М в автомат.режиме
      x6MfromLevel : Bool;   // Управление затвором 6М в автомат.режиме
      x7MfromLevel : Bool;   // Управление затвором 7М в автомат.режиме
      x8MfromLevel : Bool;   // Управление затвором 8М в автомат.режиме
      wWord02 : Word;
      wWord03 : Word;
      wWord04 : Word;
      wFrom2to1 : UInt;   // Инкремент каждые 0.5сек для состояния связи
   END_VAR
BEGIN
END_DATA_BLOCK

// folder: InstanceDB

DATA_BLOCK "DymAI_Fault"   // DB99
{ S7_Optimized_Access := 'TRUE' }
VERSION : 0.1
// stored: InstanceOfName 1FB_DymAI_Fault
"1FB_DymAI_Fault"
BEGIN
END_DATA_BLOCK

DATA_BLOCK "SysScale_01"   // DB201
{ S7_Optimized_Access := 'TRUE' }
VERSION : 0.1
// stored: InstanceOfName 1FB_Scale
"1FB_Scale"
BEGIN
END_DATA_BLOCK

DATA_BLOCK "SysScale_02"   // DB202
{ S7_Optimized_Access := 'TRUE' }
VERSION : 0.1
// stored: InstanceOfName 1FB_Scale
"1FB_Scale"
BEGIN
END_DATA_BLOCK

DATA_BLOCK "SysScale_03"   // DB203
{ S7_Optimized_Access := 'TRUE' }
VERSION : 0.1
// stored: InstanceOfName 1FB_Scale
"1FB_Scale"
BEGIN
END_DATA_BLOCK

DATA_BLOCK "SysScale_04"   // DB204
{ S7_Optimized_Access := 'TRUE' }
VERSION : 0.1
// stored: InstanceOfName 1FB_Scale
"1FB_Scale"
BEGIN
END_DATA_BLOCK

DATA_BLOCK "SysScale_05"   // DB205
{ S7_Optimized_Access := 'TRUE' }
VERSION : 0.1
// stored: InstanceOfName 1FB_Scale
"1FB_Scale"
BEGIN
END_DATA_BLOCK

DATA_BLOCK "SysScale_06"   // DB206
{ S7_Optimized_Access := 'TRUE' }
VERSION : 0.1
// stored: InstanceOfName 1FB_Scale
"1FB_Scale"
BEGIN
END_DATA_BLOCK

DATA_BLOCK "SysScale_07"   // DB207
{ S7_Optimized_Access := 'TRUE' }
VERSION : 0.1
// stored: InstanceOfName 1FB_Scale
"1FB_Scale"
BEGIN
END_DATA_BLOCK

DATA_BLOCK "SysScale_08"   // DB208
{ S7_Optimized_Access := 'TRUE' }
VERSION : 0.1
// stored: InstanceOfName 1FB_Scale
"1FB_Scale"
BEGIN
END_DATA_BLOCK

DATA_BLOCK "SysScale_09"   // DB209
{ S7_Optimized_Access := 'TRUE' }
VERSION : 0.1
// stored: InstanceOfName 1FB_Scale
"1FB_Scale"
BEGIN
END_DATA_BLOCK

DATA_BLOCK "SysScale_10"   // DB210
{ S7_Optimized_Access := 'TRUE' }
VERSION : 0.1
// stored: InstanceOfName 1FB_Scale
"1FB_Scale"
BEGIN
END_DATA_BLOCK

DATA_BLOCK "SysScale_11"   // DB211
{ S7_Optimized_Access := 'TRUE' }
VERSION : 0.1
// stored: InstanceOfName 1FB_Scale
"1FB_Scale"
BEGIN
END_DATA_BLOCK

DATA_BLOCK "SysScale_12"   // DB212
{ S7_Optimized_Access := 'TRUE' }
VERSION : 0.1
// stored: InstanceOfName 1FB_Scale
"1FB_Scale"
BEGIN
END_DATA_BLOCK

DATA_BLOCK "SysScale_13"   // DB213
{ S7_Optimized_Access := 'TRUE' }
VERSION : 0.1
// stored: InstanceOfName 1FB_Scale
"1FB_Scale"
BEGIN
END_DATA_BLOCK

DATA_BLOCK "SysScale_14"   // DB214
{ S7_Optimized_Access := 'TRUE' }
VERSION : 0.1
// stored: InstanceOfName 1FB_Scale
"1FB_Scale"
BEGIN
END_DATA_BLOCK

DATA_BLOCK "SysScale_15"   // DB215
{ S7_Optimized_Access := 'TRUE' }
VERSION : 0.1
// stored: InstanceOfName 1FB_Scale
"1FB_Scale"
BEGIN
END_DATA_BLOCK

DATA_BLOCK "SysScale_16"   // DB216
{ S7_Optimized_Access := 'TRUE' }
VERSION : 0.1
// stored: InstanceOfName 1FB_Scale
"1FB_Scale"
BEGIN
END_DATA_BLOCK

DATA_BLOCK "SysScale_17"   // DB217
{ S7_Optimized_Access := 'TRUE' }
VERSION : 0.1
// stored: InstanceOfName 1FB_Scale
"1FB_Scale"
BEGIN
END_DATA_BLOCK

DATA_BLOCK "SysScale_18"   // DB218
{ S7_Optimized_Access := 'TRUE' }
VERSION : 0.1
// stored: InstanceOfName 1FB_Scale
"1FB_Scale"
BEGIN
END_DATA_BLOCK

DATA_BLOCK "SysScale_19"   // DB219
{ S7_Optimized_Access := 'TRUE' }
VERSION : 0.1
// stored: InstanceOfName 1FB_Scale
"1FB_Scale"
BEGIN
END_DATA_BLOCK

DATA_BLOCK "SysScale_20"   // DB220
{ S7_Optimized_Access := 'TRUE' }
VERSION : 0.1
// stored: InstanceOfName 1FB_Scale
"1FB_Scale"
BEGIN
END_DATA_BLOCK

DATA_BLOCK "SysScale_21"   // DB221
{ S7_Optimized_Access := 'TRUE' }
VERSION : 0.1
// stored: InstanceOfName 1FB_Scale
"1FB_Scale"
BEGIN
END_DATA_BLOCK

DATA_BLOCK "SysScale_22"   // DB222
{ S7_Optimized_Access := 'TRUE' }
VERSION : 0.1
// stored: InstanceOfName 1FB_Scale
"1FB_Scale"
BEGIN
END_DATA_BLOCK

DATA_BLOCK "SysScale_23"   // DB223
{ S7_Optimized_Access := 'TRUE' }
VERSION : 0.1
// stored: InstanceOfName 1FB_Scale
"1FB_Scale"
BEGIN
END_DATA_BLOCK

DATA_BLOCK "SysScale_24"   // DB224
{ S7_Optimized_Access := 'TRUE' }
VERSION : 0.1
// stored: InstanceOfName 1FB_Scale
"1FB_Scale"
BEGIN
END_DATA_BLOCK

DATA_BLOCK "SysScale_25"   // DB225
{ S7_Optimized_Access := 'TRUE' }
VERSION : 0.1
// stored: InstanceOfName 1FB_ScaleRTD
"1FB_ScaleRTD"
BEGIN
END_DATA_BLOCK

DATA_BLOCK "SysScale_26"   // DB226
{ S7_Optimized_Access := 'TRUE' }
VERSION : 0.1
// stored: InstanceOfName 1FB_ScaleRTD
"1FB_ScaleRTD"
BEGIN
END_DATA_BLOCK

DATA_BLOCK "SysScale_27"   // DB227
{ S7_Optimized_Access := 'TRUE' }
VERSION : 0.1
// stored: InstanceOfName 1FB_ScaleRTD
"1FB_ScaleRTD"
BEGIN
END_DATA_BLOCK

DATA_BLOCK "SysScale_28"   // DB228
{ S7_Optimized_Access := 'TRUE' }
VERSION : 0.1
// stored: InstanceOfName 1FB_ScaleRTD
"1FB_ScaleRTD"
BEGIN
END_DATA_BLOCK

DATA_BLOCK "SysScale_29"   // DB229
{ S7_Optimized_Access := 'TRUE' }
VERSION : 0.1
// stored: InstanceOfName 1FB_ScaleRTD
"1FB_ScaleRTD"
BEGIN
END_DATA_BLOCK

DATA_BLOCK "SysScale_30"   // DB230
{ S7_Optimized_Access := 'TRUE' }
VERSION : 0.1
// stored: InstanceOfName 1FB_ScaleRTD
"1FB_ScaleRTD"
BEGIN
END_DATA_BLOCK

DATA_BLOCK "SysScale_31"   // DB231
{ S7_Optimized_Access := 'TRUE' }
VERSION : 0.1
// stored: InstanceOfName 1FB_ScaleRTD
"1FB_ScaleRTD"
BEGIN
END_DATA_BLOCK

DATA_BLOCK "SysScale_32"   // DB232
{ S7_Optimized_Access := 'TRUE' }
VERSION : 0.1
// stored: InstanceOfName 1FB_ScaleRTD
"1FB_ScaleRTD"
BEGIN
END_DATA_BLOCK

DATA_BLOCK "SysScale_33"   // DB233
{ S7_Optimized_Access := 'TRUE' }
VERSION : 0.1
// stored: InstanceOfName 1FB_ScaleRTD
"1FB_ScaleRTD"
BEGIN
END_DATA_BLOCK

DATA_BLOCK "SysScale_34"   // DB234
{ S7_Optimized_Access := 'TRUE' }
VERSION : 0.1
// stored: InstanceOfName 1FB_ScaleRTD
"1FB_ScaleRTD"
BEGIN
END_DATA_BLOCK

DATA_BLOCK "SysScale_35"   // DB235
{ S7_Optimized_Access := 'TRUE' }
VERSION : 0.1
// stored: InstanceOfName 1FB_ScaleRTD
"1FB_ScaleRTD"
BEGIN
END_DATA_BLOCK

DATA_BLOCK "SysScale_36"   // DB236
{ S7_Optimized_Access := 'TRUE' }
VERSION : 0.1
// stored: InstanceOfName 1FB_ScaleRTD
"1FB_ScaleRTD"
BEGIN
END_DATA_BLOCK

DATA_BLOCK "SysScale_37"   // DB237
{ S7_Optimized_Access := 'TRUE' }
VERSION : 0.1
// stored: InstanceOfName 1FB_ScaleRTD
"1FB_ScaleRTD"
BEGIN
END_DATA_BLOCK

DATA_BLOCK "SysScale_38"   // DB238
{ S7_Optimized_Access := 'TRUE' }
VERSION : 0.1
// stored: InstanceOfName 1FB_ScaleRTD
"1FB_ScaleRTD"
BEGIN
END_DATA_BLOCK

DATA_BLOCK "SysScale_39"   // DB239
{ S7_Optimized_Access := 'TRUE' }
VERSION : 0.1
// stored: InstanceOfName 1FB_ScaleRTD
"1FB_ScaleRTD"
BEGIN
END_DATA_BLOCK

DATA_BLOCK "SysScale_40"   // DB240
{ S7_Optimized_Access := 'TRUE' }
VERSION : 0.1
// stored: InstanceOfName 1FB_ScaleRTD
"1FB_ScaleRTD"
BEGIN
END_DATA_BLOCK

DATA_BLOCK "Control_01"   // DB301
{ S7_Optimized_Access := 'TRUE' }
VERSION : 0.1
// stored: InstanceOfName 1FB_Control
"1FB_Control"
BEGIN
END_DATA_BLOCK

DATA_BLOCK "Control_02"   // DB302
{ S7_Optimized_Access := 'TRUE' }
VERSION : 0.1
// stored: InstanceOfName 1FB_Control
"1FB_Control"
BEGIN
END_DATA_BLOCK

DATA_BLOCK "Control_03"   // DB303
{ S7_Optimized_Access := 'TRUE' }
VERSION : 0.1
// stored: InstanceOfName 1FB_Control
"1FB_Control"
BEGIN
END_DATA_BLOCK

DATA_BLOCK "Control_04"   // DB304
{ S7_Optimized_Access := 'TRUE' }
VERSION : 0.1
// stored: InstanceOfName 1FB_Control
"1FB_Control"
BEGIN
END_DATA_BLOCK

DATA_BLOCK "Control_05"   // DB305
{ S7_Optimized_Access := 'TRUE' }
VERSION : 0.1
// stored: InstanceOfName 1FB_Control
"1FB_Control"
BEGIN
END_DATA_BLOCK

DATA_BLOCK "Control_06"   // DB306
{ S7_Optimized_Access := 'TRUE' }
VERSION : 0.1
// stored: InstanceOfName 1FB_Control
"1FB_Control"
BEGIN
END_DATA_BLOCK

DATA_BLOCK "Control_07"   // DB307
{ S7_Optimized_Access := 'TRUE' }
VERSION : 0.1
// stored: InstanceOfName 1FB_Control
"1FB_Control"
BEGIN
END_DATA_BLOCK

DATA_BLOCK "Control_08"   // DB308
{ S7_Optimized_Access := 'TRUE' }
VERSION : 0.1
// stored: InstanceOfName 1FB_Control
"1FB_Control"
BEGIN
END_DATA_BLOCK

DATA_BLOCK "Control_09"   // DB309
{ S7_Optimized_Access := 'TRUE' }
VERSION : 0.1
// stored: InstanceOfName 1FB_Control
"1FB_Control"
BEGIN
END_DATA_BLOCK

DATA_BLOCK "Control_10"   // DB310
{ S7_Optimized_Access := 'TRUE' }
VERSION : 0.1
// stored: InstanceOfName 1FB_Control
"1FB_Control"
BEGIN
END_DATA_BLOCK

DATA_BLOCK "Control_11"   // DB311
{ S7_Optimized_Access := 'TRUE' }
VERSION : 0.1
// stored: InstanceOfName 1FB_Control
"1FB_Control"
BEGIN
END_DATA_BLOCK

DATA_BLOCK "Control_12"   // DB312
{ S7_Optimized_Access := 'TRUE' }
VERSION : 0.1
// stored: InstanceOfName 1FB_Control
"1FB_Control"
BEGIN
END_DATA_BLOCK

DATA_BLOCK "Control_13"   // DB313
{ S7_Optimized_Access := 'TRUE' }
VERSION : 0.1
// stored: InstanceOfName 1FB_Control
"1FB_Control"
BEGIN
END_DATA_BLOCK

DATA_BLOCK "Control_14"   // DB314
{ S7_Optimized_Access := 'TRUE' }
VERSION : 0.1
// stored: InstanceOfName 1FB_Control
"1FB_Control"
BEGIN
END_DATA_BLOCK

DATA_BLOCK "Control_15"   // DB315
{ S7_Optimized_Access := 'TRUE' }
VERSION : 0.1
// stored: InstanceOfName 1FB_Control
"1FB_Control"
BEGIN
END_DATA_BLOCK

DATA_BLOCK "Control_16"   // DB316
{ S7_Optimized_Access := 'TRUE' }
VERSION : 0.1
// stored: InstanceOfName 1FB_Control
"1FB_Control"
BEGIN
END_DATA_BLOCK

DATA_BLOCK "Control_17"   // DB317
{ S7_Optimized_Access := 'TRUE' }
VERSION : 0.1
// stored: InstanceOfName 1FB_Control
"1FB_Control"
BEGIN
END_DATA_BLOCK

DATA_BLOCK "Control_18"   // DB318
{ S7_Optimized_Access := 'TRUE' }
VERSION : 0.1
// stored: InstanceOfName 1FB_Control
"1FB_Control"
BEGIN
END_DATA_BLOCK

DATA_BLOCK "Control_19"   // DB319
{ S7_Optimized_Access := 'TRUE' }
VERSION : 0.1
// stored: InstanceOfName 1FB_Control
"1FB_Control"
BEGIN
END_DATA_BLOCK

DATA_BLOCK "Control_20"   // DB320
{ S7_Optimized_Access := 'TRUE' }
VERSION : 0.1
// stored: InstanceOfName 1FB_Control
"1FB_Control"
BEGIN
END_DATA_BLOCK

DATA_BLOCK "Control_21"   // DB321
{ S7_Optimized_Access := 'TRUE' }
VERSION : 0.1
// stored: InstanceOfName 1FB_Control
"1FB_Control"
BEGIN
END_DATA_BLOCK

DATA_BLOCK "Control_25"   // DB325
{ S7_Optimized_Access := 'TRUE' }
VERSION : 0.1
// stored: InstanceOfName 1FB_Control
"1FB_Control"
BEGIN
END_DATA_BLOCK

DATA_BLOCK "Control_26"   // DB326
{ S7_Optimized_Access := 'TRUE' }
VERSION : 0.1
// stored: InstanceOfName 1FB_Control
"1FB_Control"
BEGIN
END_DATA_BLOCK

DATA_BLOCK "Control_27"   // DB327
{ S7_Optimized_Access := 'TRUE' }
VERSION : 0.1
// stored: InstanceOfName 1FB_Control
"1FB_Control"
BEGIN
END_DATA_BLOCK

DATA_BLOCK "Control_28"   // DB328
{ S7_Optimized_Access := 'TRUE' }
VERSION : 0.1
// stored: InstanceOfName 1FB_Control
"1FB_Control"
BEGIN
END_DATA_BLOCK

DATA_BLOCK "Control_29"   // DB329
{ S7_Optimized_Access := 'TRUE' }
VERSION : 0.1
// stored: InstanceOfName 1FB_Control
"1FB_Control"
BEGIN
END_DATA_BLOCK

DATA_BLOCK "Control_30"   // DB330
{ S7_Optimized_Access := 'TRUE' }
VERSION : 0.1
// stored: InstanceOfName 1FB_Control
"1FB_Control"
BEGIN
END_DATA_BLOCK

DATA_BLOCK "Control_31"   // DB331
{ S7_Optimized_Access := 'TRUE' }
VERSION : 0.1
// stored: InstanceOfName 1FB_Control
"1FB_Control"
BEGIN
END_DATA_BLOCK

DATA_BLOCK "Control_32"   // DB332
{ S7_Optimized_Access := 'TRUE' }
VERSION : 0.1
// stored: InstanceOfName 1FB_Control
"1FB_Control"
BEGIN
END_DATA_BLOCK

DATA_BLOCK "Control_33"   // DB333
{ S7_Optimized_Access := 'TRUE' }
VERSION : 0.1
// stored: InstanceOfName 1FB_Control
"1FB_Control"
BEGIN
END_DATA_BLOCK

DATA_BLOCK "Control_34"   // DB334
{ S7_Optimized_Access := 'TRUE' }
VERSION : 0.1
// stored: InstanceOfName 1FB_Control
"1FB_Control"
BEGIN
END_DATA_BLOCK

DATA_BLOCK "Control_35"   // DB335
{ S7_Optimized_Access := 'TRUE' }
VERSION : 0.1
// stored: InstanceOfName 1FB_Control
"1FB_Control"
BEGIN
END_DATA_BLOCK

DATA_BLOCK "Control_36"   // DB336
{ S7_Optimized_Access := 'TRUE' }
VERSION : 0.1
// stored: InstanceOfName 1FB_Control
"1FB_Control"
BEGIN
END_DATA_BLOCK

DATA_BLOCK "Control_37"   // DB337
{ S7_Optimized_Access := 'TRUE' }
VERSION : 0.1
// stored: InstanceOfName 1FB_Control
"1FB_Control"
BEGIN
END_DATA_BLOCK

DATA_BLOCK "Control_38"   // DB338
{ S7_Optimized_Access := 'TRUE' }
VERSION : 0.1
// stored: InstanceOfName 1FB_Control
"1FB_Control"
BEGIN
END_DATA_BLOCK

DATA_BLOCK "Control_39"   // DB339
{ S7_Optimized_Access := 'TRUE' }
VERSION : 0.1
// stored: InstanceOfName 1FB_Control
"1FB_Control"
BEGIN
END_DATA_BLOCK

DATA_BLOCK "Control_41"   // DB341
{ S7_Optimized_Access := 'TRUE' }
VERSION : 0.1
// stored: InstanceOfName 1FB_Control
"1FB_Control"
BEGIN
END_DATA_BLOCK

DATA_BLOCK "Control_42"   // DB342
{ S7_Optimized_Access := 'TRUE' }
VERSION : 0.1
// stored: InstanceOfName 1FB_Control
"1FB_Control"
BEGIN
END_DATA_BLOCK

DATA_BLOCK "iDBfor1M"   // DB401
{ S7_Optimized_Access := 'TRUE' }
VERSION : 0.1
// stored: InstanceOfName Control1M
"Control1M"
BEGIN
END_DATA_BLOCK

DATA_BLOCK "iDBfor2M"   // DB402
{ S7_Optimized_Access := 'TRUE' }
VERSION : 0.1
// stored: InstanceOfName Control2M
"Control2M"
BEGIN
END_DATA_BLOCK

DATA_BLOCK "iDBfor3M"   // DB403
{ S7_Optimized_Access := 'TRUE' }
VERSION : 0.1
// stored: InstanceOfName ControlGate
"ControlGate"
BEGIN
END_DATA_BLOCK

DATA_BLOCK "iDBfor4M"   // DB404
{ S7_Optimized_Access := 'TRUE' }
VERSION : 0.1
// stored: InstanceOfName ControlGate
"ControlGate"
BEGIN
END_DATA_BLOCK

DATA_BLOCK "iDBfor5M"   // DB405
{ S7_Optimized_Access := 'TRUE' }
VERSION : 0.1
// stored: InstanceOfName ControlGate
"ControlGate"
BEGIN
END_DATA_BLOCK

DATA_BLOCK "iDBfor6M"   // DB406
{ S7_Optimized_Access := 'TRUE' }
VERSION : 0.1
// stored: InstanceOfName ControlGate
"ControlGate"
BEGIN
END_DATA_BLOCK

DATA_BLOCK "iDBfor7M"   // DB407
{ S7_Optimized_Access := 'TRUE' }
VERSION : 0.1
// stored: InstanceOfName ControlGate
"ControlGate"
BEGIN
END_DATA_BLOCK

DATA_BLOCK "iDBfor8M"   // DB408
{ S7_Optimized_Access := 'TRUE' }
VERSION : 0.1
// stored: InstanceOfName ControlGate
"ControlGate"
BEGIN
END_DATA_BLOCK

DATA_BLOCK "iDBforDym"   // DB409
{ S7_Optimized_Access := 'TRUE' }
VERSION : 0.1
// stored: InstanceOfName ControlDym
"ControlDym"
BEGIN
END_DATA_BLOCK

// folder: Machinery

DATA_BLOCK "CommTest_DB"   // DB98
{ S7_Optimized_Access := 'TRUE' }
VERSION : 0.1
// stored: InstanceOfName 1FB_CommTest
"1FB_CommTest"
BEGIN
END_DATA_BLOCK

DATA_BLOCK "HMI-Machinery"   // DB501
{ S7_Optimized_Access := 'FALSE' }
VERSION : 0.1
   VAR
      "1M" : "uHMI-Machine";
      "1M_PID" : "uHMI-PID";
      "2M" : "uHMI-Machine";
      Dym : "uHMI-Dym";
      Dym_PID : "uHMI-PID";
      Spare11 : Real;
      Spare12 : Real;
      Spare13 : Real;
      Spare14 : Real;
      Spare15 : Real;
      xButtonAckAll : Bool;   // Сброс всех аварий одной кнопкой
      xButtTotalSTOP : Bool;   // Функциональный останов
      xButSirenOff : Bool;   // Кнопка выключения звука
      xFaDymCummHMI : Bool;   // Бит ЧМИ остановки дымососа по аварии одного и более датчиков
      xFaDymSensors : Bool;   // Бит остановки дымососа по аварии одного и более датчиков
      "xSpare190.5" : Bool;
      xAlarmSirenOn : Bool;   // Звуковая сигнализация включена
      xAlarmLampOn : Bool;   // Световая сигнализация включена
      wSpare192 : Word;
      wSpare194 : Word;
      wSpare196 : Word;
      usiBackCountMin : USInt;   // Осталось минут до выключения дымососа
      usiBackCountSec : USInt;   // Осталось секунд до выключения дымососа
      usiBC_ResrartMin : USInt;   // Осталось минут до разрешения включения дымососа
      usiBC_ResrartSec : USInt;   // Осталось секунд до разрешения включения дымососа
      usiSpare202 : USInt;
      usiSpare203 : USInt;
      usiSpare204 : USInt;
      usiSpare205 : USInt;
      usiSpare206 : USInt;
      usiSpare207 : USInt;
      usiSpare208 : USInt;
      usiSpare209 : USInt;
      xButtSave : Bool;   // Кнопка Сохранить настройки
      xButtRestore : Bool;   // Кнопка Возврат настроек
      xFrontSave : Bool;   // Обнаружение фронта
      xFrontRestore : Bool;   // Обнаружение фронта
   END_VAR
BEGIN
   "1M_PID".rSetpoint := 190.0;
   Dym_PID.rSetpoint := 3.0;
   "1M_PID".rProportionalGain := 1.0;
   Dym_PID.rProportionalGain := 2.0;
   Dym.iMaxStart := 3;
END_DATA_BLOCK

// folder: Machinery/Gates

DATA_BLOCK "HMI-3M"   // DB503
{ S7_Optimized_Access := 'FALSE' }
VERSION : 0.1
   VAR
      "3M" : "uHMI-Machine";
      wSpare30 : Word;
      wSpare31 : Word;
      wSpare32 : Word;
      wSpare33 : Word;
      wSpare34 : Word;
      wSpare35 : Word;
      wSpare36 : Word;
      wSpare37 : Word;
      wSpare38 : Word;
      wSpare39 : Word;
      xSpare500 : Bool;
      xSpare501 : Bool;
      xSpare502 : Bool;
      xSpare503 : Bool;
      xSpare504 : Bool;
      xSpare505 : Bool;
      xSpare506 : Bool;
      xSpare507 : Bool;
      xSpare510 : Bool;
      xSpare511 : Bool;
      xSpare512 : Bool;
      xSpare513 : Bool;
      xSpare514 : Bool;
      xSpare515 : Bool;
      xCommOK : Bool;   // Межконтроллерный обмен OK
      xCommFault : Bool;   // Отказ межконтроллерного обмена
   END_VAR
BEGIN
END_DATA_BLOCK

DATA_BLOCK "HMI-4M"   // DB504
{ S7_Optimized_Access := 'FALSE' }
VERSION : 0.1
   VAR
      "4M" : "uHMI-Machine";
   END_VAR
BEGIN
END_DATA_BLOCK

DATA_BLOCK "HMI-5M"   // DB505
{ S7_Optimized_Access := 'FALSE' }
VERSION : 0.1
   VAR
      "5M" : "uHMI-Machine";
   END_VAR
BEGIN
END_DATA_BLOCK

DATA_BLOCK "HMI-6M"   // DB506
{ S7_Optimized_Access := 'FALSE' }
VERSION : 0.1
   VAR
      "6M" : "uHMI-Machine";
   END_VAR
BEGIN
END_DATA_BLOCK

DATA_BLOCK "HMI-7M"   // DB507
{ S7_Optimized_Access := 'FALSE' }
VERSION : 0.1
   VAR
      "7M" : "uHMI-Machine";
   END_VAR
BEGIN
END_DATA_BLOCK

DATA_BLOCK "HMI-8M"   // DB508
{ S7_Optimized_Access := 'FALSE' }
VERSION : 0.1
   VAR
      "8M" : "uHMI-Machine";
   END_VAR
BEGIN
END_DATA_BLOCK

// folder: Mirrors

DATA_BLOCK "1DB_mirror_aiw"   // DB101
{ S7_Optimized_Access := 'FALSE' }
VERSION : 0.1
   VAR
      aiw_PIT201a : Int;   // Код АЦП PIT201a. Разряжение на газоходе перед циклоном
      aiw_PIT202a : Int;   // Код АЦП PIT202a. Разрежение на газохоже перед рукавным фильтром
      aiw_PIT203a : Int;   // Код АЦП PIT203a. Разрежение на газоходе после рукавного фильтра
      aiw_PIT204a : Int;   // Код АЦП PIT204a. Давл. на трубопроводе сж.воздуха на вх. в шатер рукавного фильтра
      aiw_QT503b_CO : Int;   // Код АЦП QT503b_CO. Концентрация CO
      aiw_QT503b_SO2 : Int;   // Код АЦП QT503b_SO2. Концентрация SO2
      aiw_QT503b_NOx : Int;   // Код АЦП QT503b_NOx. Концентрация NOx
      aiw_QT503b_CO2 : Int;   // Код АЦП QT503b_CO2. Концентрация CO2
      aiw_QT503b_O2 : Int;   // Код АЦП QT503b_O2. Концентрация O2
      aiw_QT303b : Int;   // Код АЦП QT303b. Расход пылегазовой смеси
      aiw_QT403b : Int;   // Код АЦП QT403b. Концентрация пыли
      aiw_PV1M : Int;   // Код АЦП PV1M. Положение: клапан регулирующий для аспирации 1M
      aiw_IT1 : Int;   // Код АЦП IT1. Контроль тока двигателя (Шкаф ШПЧ1)
      aiw_RT1 : Int;   // Код АЦП RT1. Контроль скорости (Шкаф ШПЧ1)
      Spare28 : Int;   // Резерв
      Spare30 : Int;   // Резерв
      aiw_VE801a : Int;   // Код АЦП VE801a. Дымосос 1. Вибрация переднего подшипника вентилятора X-направления
      aiw_VE802a : Int;   // Код АЦП VE802a. Дымосос 1. Вибрация переднего подшипника вентилятора Y-направления
      aiw_VE803a : Int;   // Код АЦП VE803a. Дымосос 1. Вибрация заднего подшипника вентилятора X-направления
      aiw_VE804a : Int;   // Код АЦП VE804a. Дымосос 1. Вибрация заднего подшипника вентилятора Y-направления
      Spare40 : Int;   // Резерв
      Spare42 : Int;   // Резерв
      Spare44 : Int;   // Резерв
      Spare46 : Int;   // Резерв
      aiw_TE104a : Int;   // Код АЦП TE104a. Дымосос 1. Температура переднего подшипника вентилятора
      aiw_TE105a : Int;   // Код АЦП TE105a. Дымосос 1. Температура заднего подшипника вентилятора
      aiw_TE106a : Int;   // Код АЦП TE106a. Электродвигатель дымососа 1. Температура переднего подшипника
      aiw_TE107a : Int;   // Код АЦП TE107a. Электродвигатель дымососа 1. Температура заднего подшипника
      aiw_TE108a : Int;   // Код АЦП TE108a. Электродвигатель дымососа 1. Температура обмотки А
      aiw_TE109a : Int;   // Код АЦП TE109a. Электродвигатель дымососа 1. Температура обмотки А'
      aiw_TE110a : Int;   // Код АЦП TE110a. Электродвигатель дымососа 1. Температура обмотки B
      aiw_TE111a : Int;   // Код АЦП TE111a. Электродвигатель дымососа 1. Температура обмотки B
      aiw_TE112a : Int;   // Код АЦП TE112a. Электродвигатель дымососа 1. Температура обмотки C
      aiw_TE113a : Int;   // Код АЦП TE113a. Электродвигатель дымососа 1. Температура обмотки C'
      Spare68 : Int;   // Резерв
      Spare70 : Int;   // Резерв
      aiw_TE101a : Int;   // Код АЦП TE101a. Температура на газоходе перед циклоном
      aiw_TE102a : Int;   // Код АЦП TE102a. Температура на газоходе перед рукавным фильтром
      aiw_TE103a : Int;   // Код АЦП TE103a. Температура газа на выходе из трубы
      iSpare78 : Int;   // Резерв
      iSpare80 : Int;   // Резерв
      iSpare82 : Int;   // Резерв
      iSpare83 : Int;   // Резерв
      iSpare84 : Int;   // Резерв
      iSpare85 : Int;   // Резерв
      iSpare86 : Int;   // Резерв
      iSpare87 : Int;   // Резерв
      iSpare88 : Int;   // Резерв
      "iTest4-20" : Int;   // Тестируем алгоритмы Аналогового входа 4-20mA
      iTestRTD : Int;   // Тестируем алгоритмы Аналогового входа RTD (термометр)
   END_VAR
BEGIN
END_DATA_BLOCK

DATA_BLOCK "1DB_mirror_di"   // DB102
{ S7_Optimized_Access := 'FALSE' }
VERSION : 0.1
   VAR
      di_2KV1 : Bool;   // Направляющий аппарат 2М. Напряжение подано
      di_2KV4 : Bool;   // Направляющий аппарат 2М. Выбран режим ДУ
      di_2KM : Bool;   // Направляющий аппарат 2М. Сигнал РАБОТА
      di_2KV2 : Bool;   // Направляющий аппарат 2М. ОТКРЫТ
      di_2KV3 : Bool;   // Направляющий аппарат 2М. ЗАКРЫТ
      di_3KV1 : Bool;   // Затвор шлюзовый 3М. Напряжение подано
      di_3KV2 : Bool;   // Затвор шлюзовый 3М. Выбран режим ДУ
      di_3KM1 : Bool;   // Затвор шлюзовый 3М. Сигнал РАБОТА
      di_1KV8 : Bool;   // Клапан регулирующий для аспирации 1М. Напряжение подано
      di_1KV6 : Bool;   // Клапан регулирующий для аспирации 1М. Выбран режим ДУ
      di_1KM1_1KV8 : Bool;   // Клапан регулирующий для аспирации 1М. Сигнал ГОТОВНОСТЬ
      di_1KV3 : Bool;   // Клапан регулирующий для аспирации 1М. Полностью ОТКРЫТ
      di_1KV4 : Bool;   // Клапан регулирующий для аспирации 1М. Полностью ЗАКРЫТ
      di_4KV1 : Bool;   // Затвор шлюзовый 4М. Напряжение подано
      di_4KV2 : Bool;   // Затвор шлюзовый 4М. Выбран режим ДУ
      di_4KM1 : Bool;   // Затвор шлюзовый 4М. Сигнал РАБОТА
      di_5KV1 : Bool;   // Затвор шлюзовый 5М. Напряжение подано
      di_5KV2 : Bool;   // Затвор шлюзовый 5М. Режим ДУ
      di_5KM1 : Bool;   // Затвор шлюзовый 5М. Сигнал РАБОТА
      di_6KV1 : Bool;   // Затвор шлюзовый 6М. Напряжение подано
      di_6KV2 : Bool;   // Затвор шлюзовый 6М. Режим ДУ
      di_6KM1 : Bool;   // Затвор шлюзовый 6М. Сигнал РАБОТА
      "Spare2.6" : Bool;
      "Spare2.7" : Bool;
      di_7KV1 : Bool;   // Затвор шлюзовый 7М. Напряжение подано
      di_7KV2 : Bool;   // Затвор шлюзовый 7М. Режим ДУ
      di_7KM1 : Bool;   // Затвор шлюзовый 7М. Сигнал РАБОТА
      di_8KV1 : Bool;   // Затвор шлюзовый 8М. Напряжение подано
      di_8KV2 : Bool;   // Затвор шлюзовый 8М. Режим ДУ
      di_8KM1 : Bool;   // Затвор шлюзовый 8М. Сигнал РАБОТА
      "Spare3.6" : Bool;
      "Spare3.7" : Bool;
      "di_1-5QF1" : Bool;   // Шкаф ШЭ. Ввод 1 (230В, 50Гц). Вводной выключатель ШЭ включен
      "di_1-5QF2" : Bool;   // Шкаф ШЭ. Фидер (230В, 50Гц) 1ШК ФРИР включен (питание клапанов)
      "di_1-5QF3" : Bool;   // Шкаф ШЭ. 230В, 50Гц. Выключатель ИБП выключен
      "di_1-5QF4" : Bool;   // Шкаф ШЭ. Фидер (230В, 50Гц) 1ШК ФРИР от ИБП включен (питание ПЛК, датчиков)
      "di_1-5QF5" : Bool;   // Шкаф ШЭ. Фидер (230В, 50Гц) 1ШК ГО от ИБП включен
      "di_1-5QF6" : Bool;   // Шкаф ШЭ. Фидер (230В, 50Гц) ШГМ от ИБП включен
      "di_1-5QF7" : Bool;   // Шкаф ШЭ. Фидер (230В, 50Гц) ШРС от ИБП включен
      di_5SF3 : Bool;   // Шкаф ШЭ. Вводный выключатель обогрева включен
      "di_1-5Uno" : Bool;   // Шкаф ШЭ. Контроль уровня заряда батареи. В норме
      "di_1-5Unc" : Bool;   // Шкаф ШЭ. Контроль уровня заряда батареи. Ниже допустимого
      "di_5A1-K2" : Bool;   // Шкаф ШЭ. Дверь закрыта при подкл. агрегате к питанию 230В,50Гц, контакт К2 замкнут
      "di_5A1-K1" : Bool;   // Шкаф ШЭ. Температура при подкл. агрегата к питанию 230В,50Гц в норме, контакт К1 замкнут
      di_5SF1 : Bool;   // Шкаф ШЭ. Вводной выключатель кондиционера включен
      di_1K62 : Bool;   // Шкаф 1ШК. Дверь закрыта при подкл. агрегате к питанию 230В,50Гц, контакт К2 замкнут
      di_1K63 : Bool;   // Шкаф 1ШК. Температура при подкл. агрегата к питанию 230В,50Гц в норме, контакт К1 замкнут
      "Spare5.7" : Bool;
      "di_ShPCh1-10KV1" : Bool;   // Высокое напряжение подано (Шкаф преобразователя частоты ШПЧ1)
      "di_ShPCh1-10KV2" : Bool;   // Режим МУ от ключа (Шкаф преобразователя частоты ШПЧ1)
      "di_ShPCh1-10KV5" : Bool;   // Режим ДУ от ключа (Шкаф преобразователя частоты ШПЧ1)
      "di_ShPCh1-10KV6" : Bool;   // Разрешить импульсы (Шкаф преобразователя частоты ШПЧ1)
      "di_ShPCh1-10KV7" : Bool;   // Авария=0, нет аварии=1 (Шкаф преобразователя частоты ШПЧ1)
      "di_ShPCh1-10KV11" : Bool;   // Готовность привода (Шкаф преобразователя частоты ШПЧ1)
      "di_ShPCh1-10KV13" : Bool;   // Дистанционное управление (Шкаф преобразователя частоты ШПЧ1)
      "di_ShPCh1-10KV14" : Bool;   // Местное управление (Шкаф преобразователя частоты ШПЧ1)
      Spare7 : Byte;
      "Spare8.0" : Bool;
   END_VAR
BEGIN
END_DATA_BLOCK

DATA_BLOCK "1DB_mirror_out"   // DB103
{ S7_Optimized_Access := 'FALSE' }
VERSION : 0.1
   VAR
      aow_RV1 : Int;   // Задание скорости (Шкаф преобразователя частоты ШПЧ1)
      Spare2 : Int;   // Резерв
      "Spare4.0" : Bool;   // Резерв
      "Spare4.1" : Bool;   // Резерв
      "Spare4.2" : Bool;   // Резерв
      "Spare4.3" : Bool;   // Резерв
      "Spare4.4" : Bool;   // Резерв
      "Spare4.5" : Bool;   // Резерв
      "Spare4.6" : Bool;   // Резерв
      "Spare4.7" : Bool;   // Резерв
      Spare5 : Byte;   // Резерв
      Spare6 : Byte;   // Резерв
      do_2M_Open : Bool;   // Команда ОТКРЫТЬ (Направляющий аппарат 2М)
      do_2M_Close : Bool;   // Команда ЗАКРЫТЬ (Направляющий аппарат 2М)
      do_1M_Open : Bool;   // Команда ОТКРЫТЬ (Регулирующий клапан 1М)
      do_1M_Close : Bool;   // Команда ЗАКРЫТЬ (Регулирующий клапан 1М)
      do_3KV3 : Bool;   // Команда ПУСК (Затвор шлюзовый 3М)
      do_4KV3 : Bool;   // Команда ПУСК (Затвор шлюзовый 4М)
      do_5KV3 : Bool;   // Команда ПУСК (Затвор шлюзовый 5М)
      do_6KV3 : Bool;   // Команда ПУСК (Затвор шлюзовый 6М)
      do_7KV3 : Bool;   // Команда ПУСК (Затвор шлюзовый 7М)
      do_8KV3 : Bool;   // Команда ПУСК (Затвор шлюзовый 8М)
      do_10KV9 : Bool;   // Команда ПУСК (Шкаф преобразователя частоты ШПЧ1)
      do_10KV10 : Bool;   // Команда СТОП, акт.сигнал=0 (Шкаф преобр.частоты ШПЧ1)
      "xSpare8.4" : Bool;   // Резерв
      "xSpare8.5" : Bool;   // Резерв
      do_AlarmBuzzer : Bool;   // Аварийная сигнализация, звонок
      do_AlarmLamp : Bool;   // Аварийная сигнализация, лампа
   END_VAR
BEGIN
END_DATA_BLOCK

DATA_BLOCK "1DB_ANTI_di"   // DB112
{ S7_Optimized_Access := 'FALSE' }
VERSION : 0.1
   VAR
      xSpare2 : Bool;
      xSpare3 : Bool;
      xSpare4 : Bool;
      xSpare5 : Bool;
      xSpare6 : Bool;
      xSpare7 : Bool;
      xSpare8 : Bool;
      xSpare9 : Bool;
      xSpare10 : Bool;
      xSpare11 : Bool;
      xSpare12 : Bool;
      xSpare13 : Bool;
      xSpare14 : Bool;
      xSpare15 : Bool;
      xSpare16 : Bool;
      xSpare17 : Bool;
      xSpare18 : Bool;
      xSpare19 : Bool;
      xSpare20 : Bool;
      xSpare21 : Bool;
      xSpare22 : Bool;
      xSpare23 : Bool;
      xSpare24 : Bool;
      xSpare25 : Bool;
      xSpare26 : Bool;
      xSpare27 : Bool;
      xSpare28 : Bool;
      xSpare29 : Bool;
      xSpare30 : Bool;
      xSpare31 : Bool;
      xSpare32 : Bool;
      xSpare33 : Bool;
      "di_1-5QF1" : Bool;   // Шкаф ШЭ. Ввод 1 (230В, 50Гц). Вводной выключатель ШЭ включен
      "di_1-5QF2" : Bool;   // Шкаф ШЭ. Фидер (230В, 50Гц) 1ШК ФРИР включен (питание клапанов)
      "di_1-5QF3" : Bool;   // Шкаф ШЭ. 230В, 50Гц. Выключатель ИБП выключен
      "di_1-5QF4" : Bool;   // Шкаф ШЭ. Фидер (230В, 50Гц) 1ШК ФРИР от ИБП включен (питание ПЛК, датчиков)
      "di_1-5QF5" : Bool;   // Шкаф ШЭ. Фидер (230В, 50Гц) 1ШК ГО от ИБП включен
      "di_1-5QF6" : Bool;   // Шкаф ШЭ. Фидер (230В, 50Гц) ШГМ от ИБП включен
      "di_1-5QF7" : Bool;   // Шкаф ШЭ. Фидер (230В, 50Гц) ШРС от ИБП включен
      di_5SF3 : Bool;   // Шкаф ШЭ. Вводный выключатель обогрева включен
      "di_1-5Uno" : Bool;   // Шкаф ШЭ. Контроль уровня заряда батареи. В норме
      "di_1-5Unc" : Bool;   // Шкаф ШЭ. Контроль уровня заряда батареи. Ниже допустимого
      "di_5A1-K2" : Bool;   // Шкаф ШЭ. Дверь закрыта при подкл. агрегате к питанию 230В,50Гц, контакт К2 замкнут
      "di_5A1-K1" : Bool;   // Шкаф ШЭ. Температура при подкл. агрегата к питанию 230В,50Гц в норме, контакт К1 замкнут
      di_5SF1 : Bool;   // Шкаф ШЭ. Вводной выключатель кондиционера включен
      di_1K62 : Bool;   // Шкаф 1ШК. Дверь закрыта при подкл. агрегате к питанию 230В,50Гц, контакт К2 замкнут
      di_1K63 : Bool;   // Шкаф 1ШК. Температура при подкл. агрегата к питанию 230В,50Гц в норме, контакт К1 замкнут
      "Spare5.7" : Bool;
      "di_ShPCh1-10KV1" : Bool;   // Высокое напряжение подано (Шкаф преобразователя частоты ШПЧ1)
      "di_ShPCh1-10KV2" : Bool;   // Режим МУ от ключа (Шкаф преобразователя частоты ШПЧ1)
      "di_ShPCh1-10KV5" : Bool;   // Режим ДУ от ключа (Шкаф преобразователя частоты ШПЧ1)
      "di_ShPCh1-10KV6" : Bool;   // Разрешить импульсы (Шкаф преобразователя частоты ШПЧ1)
      "di_ShPCh1-10KV7" : Bool;   // Авария=0, нет аварии=1 (Шкаф преобразователя частоты ШПЧ1)
      "di_ShPCh1-10KV11" : Bool;   // Готовность привода (Шкаф преобразователя частоты ШПЧ1)
      "di_ShPCh1-10KV13" : Bool;   // Дистанционное управление (Шкаф преобразователя частоты ШПЧ1)
      "di_ShPCh1-10KV14" : Bool;   // Местное управление (Шкаф преобразователя частоты ШПЧ1)
      Spare7 : Byte;
      "Spare8.0" : Bool;
   END_VAR
BEGIN
END_DATA_BLOCK

// folder: Processing_AIO

DATA_BLOCK "1DB_AICode"   // DB135
TITLE = Ошибки обрабовки аналоговых входов
{ S7_Optimized_Access := 'FALSE' }
VERSION : 0.1
// Блок данных ошибое для всех аналоговых входов
   VAR
      RarefactFlueInCyclone : Word;   // Разрежение на газоходе перед циклоном PIT201a
      RarefactFlueInFilter : Word;   // Разрежение на газоходе перед рукавным фильтром PIT202a
      RarefactFlueOutFilter : Word;   // Разрежение на газоходе после рукавного фильтра PIT203a
      PressureComprAir : Word;   // Давл. на трубопроводе сж.воздуха на вх. в шатер рукавного фильтра PIT204a
      GasAnalyzerCO : Word;   // Концентрация CO QT503b_CO
      GasAnalyzerSO2 : Word;   // Концентрация SO2 QT503b_SO2
      GasAnalyzerNOx : Word;   // Концентрация NOx QT503b_NOx
      GasAnalyzerCO2 : Word;   // Концентрация CO2 QT503b_CO2
      GasAnalyzerO2 : Word;   // Концентрация O2 QT503b_O2
      FlowDustGasMix : Word;   // Расход пылегазовой смеси QT303b
      GasAnalyzerDust : Word;   // Концентрация пыли QT403b
      PosValve1M : Word;   // Положение: клапан регулирующий 1M для аспирации PV1M
      CurrentMotorShPCh1 : Word;   // Контроль тока двигателя (Шкаф ШПЧ1) IT1
      RpmMotorShPCh1 : Word;   // Контроль скорости (Шкаф ШПЧ1) RT1
      D1FanVibrFrontX : Word;   // Дымосос 1. Вибрация переднего подшипника вентилятора X-направления VE801a
      D1FanVibrFrontY : Word;   // Дымосос 1. Вибрация переднего подшипника вентилятора Y-направления VE802a
      D1FanVibrBackX : Word;   // Дымосос 1. Вибрация заднего подшипника вентилятора X-направления VE803a
      D1FanVibrBackY : Word;   // Дымосос 1. Вибрация заднего подшипника вентилятора Y-направления VE804a
      D1FanTempFront : Word;   // Дымосос 1. Температура переднего подшипника вентилятора TE104a
      D1FanTempBack : Word;   // Дымосос 1. Температура заднего подшипника вентилятора TE105a
      D1MotorTempFront : Word;   // Электродвигатель дымососа 1. Температура переднего подшипника TE106a
      D1MotorTempBack : Word;   // Электродвигатель дымососа 1. Температура заднего подшипника TE107a
      D1MotorTempWindA1 : Word;   // Электродвигатель дымососа 1. Температура обмотки А TE108a
      D1MotorTempWindA2 : Word;   // Электродвигатель дымососа 1. Температура обмотки А' TE109a
      D1MotorTempWindB1 : Word;   // Электродвигатель дымососа 1. Температура обмотки B TE110a
      D1MotorTempWindB2 : Word;   // Электродвигатель дымососа 1. Температура обмотки B' TE111a
      D1MotorTempWindC1 : Word;   // Электродвигатель дымососа 1. Температура обмотки C TE112a
      D1MotorTempWindC2 : Word;   // Электродвигатель дымососа 1. Температура обмотки C' TE113a
      TGasDuctInCyclone : Word;   // Температура на газоходе перед циклоном TE101a
      TGasDuctInFilter : Word;   // Температура на газоходе перед рукавным фильтром TE102a
      TGasOutPipe : Word;   // Температура газа на выходе из трубы TE103a
      wSpare62 : Word;   // 1
      wSpare63 : Word;   // 2
      wSpare64 : Word;   // 3
      wSpare65 : Word;   // 4
      wSpare66 : Word;   // 5
      wSpare67 : Word;   // 6
      wSpare68 : Word;   // 7
      wSpare69 : Word;   // 8
      wSpare70 : Word;   // 9
      wSpare71 : Word;   // 10
      wSpare72 : Word;   // 11
      wSpare73 : Word;   // 12
      wSpare74 : Word;   // 13
      wSpare75 : Word;   // 14
      wSpare76 : Word;   // 15
      wSpare77 : Word;   // 16
      wSpare78 : Word;   // 17
      "wTest4-20" : Word;   // Тестируем алгоритмы Аналогового входа 4-20mA
      wTestRTD : Word;   // Тестируем алгоритмы Аналогового входа RTD (термометр)
      xF_PIT201a : Bool;   // Авария датчика PIT201a. Разряжение на газоходе перед циклоном
      xF_PIT202a : Bool;   // Авария датчика PIT202a. Разрежение на газохоже перед рукавным фильтром
      xF_PIT203a : Bool;   // Авария датчика PIT203a. Разрежение на газоходе после рукавного фильтра
      xF_PIT204a : Bool;   // Авария датчика PIT204a. Давл. на трубопроводе сж.воздуха на вх. в шатер рукавного фильтра
      xF_QT503b_CO : Bool;   // Авария датчика QT503b_CO. Концентрация CO
      xF_QT503b_SO2 : Bool;   // Авария датчика QT503b_SO2. Концентрация SO2
      xF_QT503b_NOx : Bool;   // Авария датчика QT503b_NOx. Концентрация NOx
      xF_QT503b_CO2 : Bool;   // Авария датчика QT503b_CO2. Концентрация CO2
      xF_QT503b_O2 : Bool;   // Авария датчика QT503b_O2. Концентрация O2
      xF_QT303b : Bool;   // Авария датчика QT303b. Расход пылегазовой смеси
      xF_QT403b : Bool;   // Авария датчика QT403b. Концентрация пыли
      xF_PV1M : Bool;   // Авария датчика PV1M. Положение: клапан регулирующий для аспирации 1M
      xF_IT1 : Bool;   // Авария датчика IT1. Контроль тока двигателя (Шкаф ШПЧ1)
      xF_RT1 : Bool;   // Авария датчика RT1. Контроль скорости (Шкаф ШПЧ1)
      Spare28 : Bool;   // Резерв
      Spare30 : Bool;   // Резерв
      xF_VE801a : Bool;   // Авария датчика VE801a. Дымосос 1. Вибрация переднего подшипника вентилятора X-направления
      xF_VE802a : Bool;   // Авария датчика VE802a. Дымосос 1. Вибрация переднего подшипника вентилятора Y-направления
      xF_VE803a : Bool;   // Авария датчика VE803a. Дымосос 1. Вибрация заднего подшипника вентилятора X-направления
      xF_VE804a : Bool;   // Авария датчика VE804a. Дымосос 1. Вибрация заднего подшипника вентилятора Y-направления
      Spare40 : Bool;   // Резерв
      Spare42 : Bool;   // Резерв
      Spare44 : Bool;   // Резерв
      Spare46 : Bool;   // Резерв
      xF_TE104a : Bool;   // Авария датчика TE104a. Дымосос 1. Температура переднего подшипника вентилятора
      xF_TE105a : Bool;   // Авария датчика TE105a. Дымосос 1. Температура заднего подшипника вентилятора
      xF_TE106a : Bool;   // Авария датчика TE106a. Электродвигатель дымососа 1. Температура переднего подшипника
      xF_TE107a : Bool;   // Авария датчика TE107a. Электродвигатель дымососа 1. Температура заднего подшипника
      xF_TE108a : Bool;   // Авария датчика TE108a. Электродвигатель дымососа 1. Температура обмотки А
      xF_TE109a : Bool;   // Авария датчика TE109a. Электродвигатель дымососа 1. Температура обмотки А'
      xF_TE110a : Bool;   // Авария датчика TE110a. Электродвигатель дымососа 1. Температура обмотки B
      xF_TE111a : Bool;   // Авария датчика TE111a. Электродвигатель дымососа 1. Температура обмотки B
      xF_TE112a : Bool;   // Авария датчика TE112a. Электродвигатель дымососа 1. Температура обмотки C
      xF_TE113a : Bool;   // Авария датчика TE113a. Электродвигатель дымососа 1. Температура обмотки C'
      "xSpare104.2" : Bool;   // Резерв
      "xSpare104.3" : Bool;   // Резерв
      xF_TE101a : Bool;   // Авария датчика TE101a. Температура на газоходе перед циклоном
      xF_TE102a : Bool;   // Авария датчика TE102a. Температура на газоходе перед рукавным фильтром
      xF_TE103a : Bool;   // Авария датчика TE103a. Температура газа на выходе из трубы
      "xSpare104.7" : Bool;   // Резерв
      "xSpare105.0" : Bool;   // Резерв
      "xSpare105.1" : Bool;   // Резерв
      "xSpare105.2" : Bool;   // Резерв
      "xSpare105.3" : Bool;   // Резерв
      "xSpare105.4" : Bool;   // Резерв
      "xSpare105.5" : Bool;   // Резерв
      "xSpare105.6" : Bool;   // Резерв
      "xSpare105.7" : Bool;   // Резерв
      "xF_Test4-20" : Bool;   // Тестируем алгоритмы Аналогового входа 4-20mA
      xF_TestRTD : Bool;   // Тестируем алгоритмы Аналогового входа RTD (термометр)
   END_VAR
BEGIN
END_DATA_BLOCK

DATA_BLOCK "SysScale_49"   // DB249
{ S7_Optimized_Access := 'TRUE' }
VERSION : 0.1
// stored: InstanceOfName 1FB_Scale
"1FB_Scale"
BEGIN
END_DATA_BLOCK

DATA_BLOCK "SysScale_50"   // DB250
{ S7_Optimized_Access := 'TRUE' }
VERSION : 0.1
// stored: InstanceOfName 1FB_ScaleRTD
"1FB_ScaleRTD"
BEGIN
END_DATA_BLOCK

DATA_BLOCK "Control_49"   // DB349
{ S7_Optimized_Access := 'TRUE' }
VERSION : 0.1
// stored: InstanceOfName 1FB_Control
"1FB_Control"
BEGIN
END_DATA_BLOCK

DATA_BLOCK "Control_50"   // DB350
{ S7_Optimized_Access := 'TRUE' }
VERSION : 0.1
// stored: InstanceOfName 1FB_Control
"1FB_Control"
BEGIN
END_DATA_BLOCK

// folder: Shadow

DATA_BLOCK "1DB_AIConfig_Sh"   // DB1006
TITLE = Конфигурация аналоговых входов
{ S7_Optimized_Access := 'FALSE' }
VERSION : 0.1
// Блок данных содержит параметры шкалы, фильтрации, признак лимитирования
   VAR
      RarefactFlueInCyclone : "uScale";   // Разрежение на газоходе перед циклоном PIT201a
      RarefactFlueInFilter : "uScale";   // Разрежение на газоходе перед рукавным фильтром PIT202a
      RarefactFlueOutFilter : "uScale";   // Разрежение на газоходе после рукавного фильтра PIT203a
      PressureComprAir : "uScale";   // Давл. на трубопроводе сж.воздуха на вх. в шатер рукавного фильтра PIT204a
      GasAnalyzerCO : "uScale";   // Концентрация CO QT503b_CO
      GasAnalyzerSO2 : "uScale";   // Концентрация SO2 QT503b_SO2
      GasAnalyzerNOx : "uScale";   // Концентрация NOx QT503b_NOx
      GasAnalyzerCO2 : "uScale";   // Концентрация CO2 QT503b_CO2.
      GasAnalyzerO2 : "uScale";   // Концентрация O2 QT503b_O2
      FlowDustGasMix : "uScale";   // Расход пылегазовой смеси QT303b
      GasAnalyzerDust : "uScale";   // Концентрация пыли QT403b
      PosValve1M : "uScale";   // Положение: клапан регулирующий 1M для аспирации PV1M.
      CurrentMotorShPCh1 : "uScale";   // Контроль тока двигателя (Шкаф ШПЧ1) IT1
      RpmMotorShPCh1 : "uScale";   // Контроль скорости (Шкаф ШПЧ1) RT1
      D1FanVibrFrontX : "uScale";   // Дымосос 1. Вибрация переднего подшипника вентилятора X-направления VE801a
      D1FanVibrFrontY : "uScale";   // Дымосос 1. Вибрация переднего подшипника вентилятора Y-направления VE802a
      D1FanVibrBackX : "uScale";   // Дымосос 1. Вибрация заднего подшипника вентилятора X-направления VE803a
      D1FanVibrBackY : "uScale";   // Дымосос 1. Вибрация заднего подшипника вентилятора Y-направления VE804a
      D1FanTempFront : "uScale";   // Дымосос 1. Температура переднего подшипника вентилятора TE104a
      D1FanTempBack : "uScale";   // Дымосос 1. Температура заднего подшипника вентилятора TE105a
      D1MotorTempFront : "uScale";   // Электродвигатель дымососа 1. Температура переднего подшипника TE106a
      D1MotorTempBack : "uScale";   // Электродвигатель дымососа 1. Температура заднего подшипника TE107a
      D1MotorTempWindA1 : "uScale";   // Электродвигатель дымососа 1. Температура обмотки А TE108a
      D1MotorTempWindA2 : "uScale";   // Электродвигатель дымососа 1. Температура обмотки А' TE109a
      D1MotorTempWindB1 : "uScale";   // Электродвигатель дымососа 1. Температура обмотки B TE110a
      D1MotorTempWindB2 : "uScale";   // Электродвигатель дымососа 1. Температура обмотки B TE111a
      D1MotorTempWindC1 : "uScale";   // Электродвигатель дымососа 1. Температура обмотки C TE112a
      D1MotorTempWindC2 : "uScale";   // Электродвигатель дымососа 1. Температура обмотки C' TE113a
      TGasDuctInCyclone : "uScale";   // Температура на газоходе перед циклоном TE101a
      TGasDuctInFilter : "uScale";   // Температура на газоходе перед рукавным фильтром TE102a
      TGasOutPipe : "uScale";   // Температура газа на выходе из трубы TE103a
      uSpare558 : "uScale";   // 1
      uSpare559 : "uScale";   // 2
      uSpare560 : "uScale";   // 3
      uSpare561 : "uScale";   // 4
      uSpare562 : "uScale";   // 5
      uSpare563 : "uScale";   // 6
      uSpare564 : "uScale";   // 7
      uSpare565 : "uScale";   // 8
      uSpare566 : "uScale";   // 9
      uSpare567 : "uScale";   // 10
   END_VAR
BEGIN
   RarefactFlueInCyclone.Qmax := 10.0;
   FlowDustGasMix.Qmax := 500.0;
   RarefactFlueInCyclone.FilterTau := 0.5;
   RarefactFlueInFilter.Qmax := 10.0;
   RarefactFlueOutFilter.Qmax := 10.0;
   PressureComprAir.Qmax := 10.0;
   GasAnalyzerCO.Qmax := 300.0;
   GasAnalyzerSO2.Qmax := 500.0;
   GasAnalyzerNOx.Qmax := 500.0;
   GasAnalyzerCO2.Qmax := 4.0;
   GasAnalyzerO2.Qmax := 20.0;
   GasAnalyzerDust.Qmax := 500.0;
   CurrentMotorShPCh1.Qmax := 906.0;
   RpmMotorShPCh1.Qmax := 991.0;
   D1FanVibrFrontX.Qmax := 20.0;
   D1FanVibrFrontY.Qmax := 20.0;
   D1FanVibrBackX.Qmax := 20.0;
   D1FanVibrBackY.Qmax := 20.0;
   D1FanTempFront.Qmax := 200.0;
   D1FanTempBack.Qmax := 200.0;
   D1MotorTempFront.Qmax := 200.0;
   D1MotorTempBack.Qmax := 200.0;
   D1MotorTempWindA1.Qmax := 200.0;
   D1MotorTempWindA2.Qmax := 200.0;
   D1MotorTempWindB1.Qmax := 200.0;
   D1MotorTempWindB2.Qmax := 200.0;
   D1MotorTempWindC1.Qmax := 200.0;
   D1MotorTempWindC2.Qmax := 200.0;
   TGasDuctInCyclone.Qmax := 350.0;
   TGasDuctInFilter.Qmax := 250.0;
   TGasOutPipe.Qmax := 250.0;
   PosValve1M.FilterON := false;
   RpmMotorShPCh1.FilterTau := 3.0;
   PressureComprAir.FilterTau := 5.0;
END_DATA_BLOCK

DATA_BLOCK "Alarm_DB_Sh"   // DB1010
TITLE = Аварийные границы
{ S7_Optimized_Access := 'FALSE' }
VERSION : 0.1
// Блок данных содержит параметры верхней и нижней аварийной границы аналоговых сигналов
   VAR
      RarefactFlueInCyclone : "uWrnngAlarm";   // Разрежение на газоходе перед циклоном PIT201a
      RarefactFlueInFilter : "uWrnngAlarm";   // Разрежение на газоходе перед рукавным фильтром PIT202a
      RarefactFlueOutFilter : "uWrnngAlarm";   // Разрежение на газоходе после рукавного фильтра PIT203a
      PressureComprAir : "uWrnngAlarm";   // Давл. на трубопроводе сж.воздуха на вх. в шатер рукавного фильтра PIT204a
      GasAnalyzerCO : "uWrnngAlarm";   // Концентрация CO QT503b_CO
      GasAnalyzerSO2 : "uWrnngAlarm";   // Концентрация SO2 QT503b_SO2
      GasAnalyzerNOx : "uWrnngAlarm";   // Концентрация NOx QT503b_NOx
      GasAnalyzerCO2 : "uWrnngAlarm";   // Концентрация CO2 QT503b_CO2.
      GasAnalyzerO2 : "uWrnngAlarm";   // Концентрация O2 QT503b_O2
      FlowDustGasMix : "uWrnngAlarm";   // Расход пылегазовой смеси QT303b
      GasAnalyzerDust : "uWrnngAlarm";   // Концентрация пыли QT403b
      PosValve1M : "uWrnngAlarm";   // Положение: клапан регулирующий 1M для аспирации PV1M.
      CurrentMotorShPCh1 : "uWrnngAlarm";   // Контроль тока двигателя (Шкаф ШПЧ1) IT1
      RpmMotorShPCh1 : "uWrnngAlarm";   // Контроль скорости (Шкаф ШПЧ1) RT1
      D1FanVibrFrontX : "uWrnngAlarm";   // Дымосос 1. Вибрация переднего подшипника вентилятора X-направления VE801a
      D1FanVibrFrontY : "uWrnngAlarm";   // Дымосос 1. Вибрация переднего подшипника вентилятора Y-направления VE802a
      D1FanVibrBackX : "uWrnngAlarm";   // Дымосос 1. Вибрация заднего подшипника вентилятора X-направления VE803a
      D1FanVibrBackY : "uWrnngAlarm";   // Дымосос 1. Вибрация заднего подшипника вентилятора Y-направления VE804a
      D1FanTempFront : "uWrnngAlarm";   // Дымосос 1. Температура переднего подшипника вентилятора TE104a
      D1FanTempBack : "uWrnngAlarm";   // Дымосос 1. Температура заднего подшипника вентилятора TE105a
      D1MotorTempFront : "uWrnngAlarm";   // Электродвигатель дымососа 1. Температура переднего подшипника TE106a
      D1MotorTempBack : "uWrnngAlarm";   // Электродвигатель дымососа 1. Температура заднего подшипника TE107a
      D1MotorTempWindA1 : "uWrnngAlarm";   // Электродвигатель дымососа 1. Температура обмотки А TE108a
      D1MotorTempWindA2 : "uWrnngAlarm";   // Электродвигатель дымососа 1. Температура обмотки А' TE109a
      D1MotorTempWindB1 : "uWrnngAlarm";   // Электродвигатель дымососа 1. Температура обмотки B TE110a
      D1MotorTempWindB2 : "uWrnngAlarm";   // Электродвигатель дымососа 1. Температура обмотки B TE111a
      D1MotorTempWindC1 : "uWrnngAlarm";   // Электродвигатель дымососа 1. Температура обмотки C TE112a
      D1MotorTempWindC2 : "uWrnngAlarm";   // Электродвигатель дымососа 1. Температура обмотки C' TE113a
      TGasDuctInCyclone : "uWrnngAlarm";   // Температура на газоходе перед циклоном TE101a
      TGasDuctInFilter : "uWrnngAlarm";   // Температура на газоходе перед рукавным фильтром TE102a
      TGasOutPipe : "uWrnngAlarm";   // Температура газа на выходе из трубы TE103a
      uSpare434 : "uWrnngAlarm";   // 1
      uSpare435 : "uWrnngAlarm";   // 2
      uSpare436 : "uWrnngAlarm";   // 3
      uSpare437 : "uWrnngAlarm";   // 4
      uSpare438 : "uWrnngAlarm";   // 5
      uSpare439 : "uWrnngAlarm";   // 6
      uSpare440 : "uWrnngAlarm";   // 7
      uSpare441 : "uWrnngAlarm";   // 8
      uSpare442 : "uWrnngAlarm";   // 9
      uSpare443 : "uWrnngAlarm";   // 10
   END_VAR
BEGIN
   RarefactFlueInCyclone.H := 5.0;
   RarefactFlueInCyclone.L := 1.0;
   RarefactFlueInFilter.H := 5.0;
   RarefactFlueInFilter.L := 1.0;
   RarefactFlueOutFilter.H := 7.0;
   RarefactFlueOutFilter.H_switch := 1;
   PressureComprAir.H := 0.9;
   PressureComprAir.L := 0.1;
   GasAnalyzerCO.H := 250.0;
   GasAnalyzerCO.H_switch := 1;
   GasAnalyzerSO2.H := 400.0;
   GasAnalyzerSO2.L := 100.0;
   GasAnalyzerNOx.H := 400.0;
   GasAnalyzerNOx.L := 100.0;
   GasAnalyzerCO2.H := 3.5;
   GasAnalyzerCO2.L := 0.5;
   GasAnalyzerO2.H := 18.0;
   GasAnalyzerO2.L := 2.0;
   FlowDustGasMix.H := 400.0;
   FlowDustGasMix.L := 100.0;
   GasAnalyzerDust.H := 400.0;
   GasAnalyzerDust.L := 100.0;
   PosValve1M.H := 90.0;
   PosValve1M.L := 10.0;
   CurrentMotorShPCh1.H := 800.0;
   CurrentMotorShPCh1.L := 100.0;
   RpmMotorShPCh1.H := 800.0;
   RpmMotorShPCh1.L := 100.0;
   D1FanVibrFrontX.H := 18.0;
   D1FanVibrFrontY.H := 18.0;
   D1FanVibrFrontY.H_switch := 1;
   D1FanVibrBackX.H := 18.0;
   D1FanVibrBackX.H_switch := 1;
   D1FanVibrBackY.H := 18.0;
   D1FanVibrBackY.H_switch := 1;
   D1FanTempFront.H := 70.0;
   D1FanTempFront.H_switch := 1;
   D1FanTempBack.H := 70.0;
   D1FanTempBack.H_switch := 1;
   D1MotorTempFront.H := 70.0;
   D1MotorTempFront.H_switch := 1;
   D1MotorTempWindC2.H := 90.0;
   D1MotorTempWindC2.H_switch := 1;
   D1MotorTempWindC1.H := 90.0;
   D1MotorTempWindC1.H_switch := 1;
   D1MotorTempWindB2.H := 90.0;
   D1MotorTempWindB2.H_switch := 1;
   D1MotorTempWindB1.H := 90.0;
   D1MotorTempWindB1.H_switch := 1;
   D1MotorTempWindA2.H := 90.0;
   D1MotorTempWindA2.H_switch := 1;
   D1MotorTempWindA1.H := 90.0;
   D1MotorTempWindA1.H_switch := 1;
   D1MotorTempBack.H := 70.0;
   D1MotorTempBack.H_switch := 1;
   TGasDuctInCyclone.H := 190.0;
   TGasDuctInCyclone.H_switch := 1;
   TGasDuctInFilter.H := 190.0;
   TGasDuctInFilter.H_switch := 1;
   TGasOutPipe.H := 700.0;
   TGasOutPipe.L := 300.0;
   D1FanVibrFrontX.H_switch := 1;
END_DATA_BLOCK

DATA_BLOCK "HMI-Machinery_Sh"   // DB1501
{ S7_Optimized_Access := 'FALSE' }
VERSION : 0.1
   VAR
      uSpare0 : "uHMI-Machine";
      "1M_PID" : "uHMI-PID";
      uSpare70 : "uHMI-Machine";
      uSpare100 : "uHMI-Dym";
      Dym_PID : "uHMI-PID";
   END_VAR
BEGIN
   "1M_PID".rSetpoint := 190.0;
   Dym_PID.rSetpoint := 3.0;
   "1M_PID".rProportionalGain := 1.0;
   Dym_PID.rProportionalGain := 2.0;
   uSpare100.iMaxStart := 3;
END_DATA_BLOCK

// folder: Simulation

DATA_BLOCK "1DB_simulation"   // DB990
{ S7_Optimized_Access := 'TRUE' }
VERSION : 0.1
   VAR
      "1M_fullOpenP" : Bool;   // Для обнаружения фронта
      "1M_fullOpenN" : Bool;   // Для обнаружения фронта
      "1M_fullCloseP" : Bool;   // Для обнаружения фронта
      "1M_fullCloseN" : Bool;   // Для обнаружения фронта
      "1M_simPos" : Bool := 1;   // Сделать 0 для выключения симуляции Позиции
      "2M_sim" : Bool := 1;   // Сделать 0 для выключения симуляции КМ
      "3M-8M_sim" : Bool := 1;   // Сделать 0 для выключения симуляции КМ
      xSpare9 : Bool;
      xSpare10 : Bool;
      xSpare11 : Bool;
      xSpare12 : Bool;
      xSpare13 : Bool;
      xSpare14 : Bool;
      xSpare15 : Bool;
      xSpare16 : Bool;
      xSpare17 : Bool;
      xSpare18 : Bool;
      xSpare19 : Bool;
      "1M_simTE102" : Bool;   // Сделать 0 для выключения симуляции т-ры
      sSpare21 : Bool;
   END_VAR
BEGIN
END_DATA_BLOCK

// folder: Simulation/SimGroup

DATA_BLOCK "1DB_sim1000"   // DB991
{ S7_Optimized_Access := 'FALSE' }
VERSION : 0.1
   VAR
      sPIT201a : "uSim";
      sPIT202a : "uSim";
      sPIT203a : "uSim";
      sPIT204a : "uSim";
      sQT503b_CO : "uSim";
      sQT503b_SO2 : "uSim";
      sQT503b_NOx : "uSim";
      sQT503b_CO2 : "uSim";
      sQT503b_O2 : "uSim";
      sQT303b : "uSim";
      sQT403b : "uSim";
      sPV1M : "uSim";
      sIT1 : "uSim";
      sRT1 : "uSim";
      Spare28 : "uSim";
      Spare30 : "uSim";
      sVE801a : "uSim";
      sVE802a : "uSim";
      sVE803a : "uSim";
      sVE804a : "uSim";
      Spare40 : "uSim";
      Spare42 : "uSim";
      Spare44 : "uSim";
      Spare46 : "uSim";
      sTE104a : "uSim";
      sTE105a : "uSim";
      sTE106a : "uSim";
      sTE107a : "uSim";
      sTE108a : "uSim";
      sTE109a : "uSim";
      sTE110a : "uSim";
      sTE111a : "uSim";
      sTE112a : "uSim";
      sTE113a : "uSim";
      Spare68 : "uSim";
      Spare70 : "uSim";
      sTE101a : "uSim";
      sTE102a : "uSim";
      sTE103a : "uSim";
      Spare78 : "uSim";
   END_VAR
BEGIN
   sPIT202a.iCounter := 15;
   sPIT201a.factor := 241.0;
   sPIT201a.offset := 194.0;
   sPIT204a.iCounter := 154;
   sPIT203a.iCounter := 314;
   sQT503b_CO.iCounter := 227;
   sQT503b_SO2.iCounter := 86;
   sQT503b_NOx.iCounter := 352;
   sQT503b_CO2.iCounter := 110;
   sQT503b_O2.iCounter := 64;
   sQT303b.iCounter := 47;
   sQT403b.iCounter := 305;
   sPV1M.iCounter := 290;
   sIT1.iCounter := 144;
   sRT1.iCounter := 169;
   sVE801a.iCounter := 33;
   sVE802a.iCounter := 177;
   sVE803a.iCounter := 106;
   sVE804a.iCounter := 28;
   sPV1M.config.auto := 0;
   sTE104a.iCounter := 5;
   sTE105a.iCounter := 97;
   sTE106a.iCounter := 300;
   sTE102a.iCounter := 350;
   sTE101a.iCounter := 209;
   Spare70.iCounter := 133;
   Spare68.iCounter := 184;
   sTE113a.iCounter := 76;
   sTE112a.iCounter := 149;
   sTE111a.iCounter := 61;
   sTE110a.iCounter := 12;
   sTE109a.iCounter := 228;
   sTE108a.iCounter := 295;
   sTE107a.iCounter := 173;
   sTE102a.config.auto := 0;
   sPIT202a.config.auto := 0;
END_DATA_BLOCK

